// TwinCAT 3 PLC project SaftyPLC
// ProgramVersion: 3.1.4026.13
// libraries:
//   Tc2_Standard, * (Beckhoff Automation GmbH)
//   Tc2_System, * (Beckhoff Automation GmbH)
//   Tc2_Utilities, * (Beckhoff Automation GmbH)
//   Tc3_Module, * (Beckhoff Automation GmbH)
// project tree:
//   DUTs/GVLs/ GVL_IO.TcGVL, GVL_Safety.TcGVL (not stored)
//   / PlcTask.TcTTO (not stored)
//   POUs/ MAIN.TcPOU
// real-time tasks:
//   TASK XTS Task: cycle T#500us, priority 1, ADS port 350
//   TASK Job Task: cycle default, priority 32
//   TASK MC-Task (MET): cycle T#2ms, priority 3, ADS port 521
//   TASK MC-Task (MPT): cycle T#10ms, priority 8, ADS port 531
//   TASK PlcTask: cycle T#500us, priority 20, ADS port 351
// I/O:
//   DEVICE Device 8 (EtherCAT), AmsNetId 0.0.0.0.9.1
//     Box 23 (AT5100-0100) [AT5100-0100 XTS XL, TwinSAFE]
//       modules: Module 1 (SAFETY)
//     Box 24 (AT5100-0100) [AT5100-0100 XTS XL, TwinSAFE]
//       modules: Module 1 (SAFETY)
//     Box 25 (AT5100-0100) [AT5100-0100 XTS XL, TwinSAFE]
//       modules: Module 1 (SAFETY)
//     Box 26 (AT5100-0100) [AT5100-0100 XTS XL, TwinSAFE]
//       modules: Module 1 (SAFETY)
//     Box 27 (AT5100-0100) [AT5100-0100 XTS XL, TwinSAFE]
//       modules: Module 1 (SAFETY)
//     Box 28 (AT5100-0100) [AT5100-0100 XTS XL, TwinSAFE]
//       modules: Module 1 (SAFETY)
//     Box 29 (AT5100-0100) [AT5100-0100 XTS XL, TwinSAFE]
//       modules: Module 1 (SAFETY)
//     Box 30 (AT5100-0100) [AT5100-0100 XTS XL, TwinSAFE]
//       modules: Module 1 (SAFETY)
//     Box 31 (AT5100-0100) [AT5100-0100 XTS XL, TwinSAFE]
//       modules: Module 1 (SAFETY)
//     Box 32 (AT5100-0100) [AT5100-0100 XTS XL, TwinSAFE]
//       modules: Module 1 (SAFETY)
//     Box 33 (AT5100-0100) [AT5100-0100 XTS XL, TwinSAFE]
//       modules: Module 1 (SAFETY)
//     Box 34 (AT5100-0100) [AT5100-0100 XTS XL, TwinSAFE]
//       modules: Module 1 (SAFETY)
//     Box 35 (AT5100-0100) [AT5100-0100 XTS XL, TwinSAFE]
//       modules: Module 1 (SAFETY)
//     Box 36 (AT5100-0100) [AT5100-0100 XTS XL, TwinSAFE]
//       modules: Module 1 (SAFETY)
//     Box 37 (AT5100-0100) [AT5100-0100 XTS XL, TwinSAFE]
//       modules: Module 1 (SAFETY)
//     Box 38 (AT5100-0100) [AT5100-0100 XTS XL, TwinSAFE]
//       modules: Module 1 (SAFETY)
//     Box 39 (AT5100-0100) [AT5100-0100 XTS XL, TwinSAFE]
//       modules: Module 1 (SAFETY)
//     Box 40 (AT5100-0100) [AT5100-0100 XTS XL, TwinSAFE]
//       modules: Module 1 (SAFETY)
//     Box 41 (AT5100-0100) [AT5100-0100 XTS XL, TwinSAFE]
//       modules: Module 1 (SAFETY)
//     Box 42 (AT5100-0100) [AT5100-0100 XTS XL, TwinSAFE]
//       modules: Module 1 (SAFETY)
//     Box 43 (AT5100-0100) [AT5100-0100 XTS XL, TwinSAFE]
//       modules: Module 1 (SAFETY)
//     Box 44 (AT5100-0100) [AT5100-0100 XTS XL, TwinSAFE]
//       modules: Module 1 (SAFETY)
//     Box 45 (AT5100-0100) [AT5100-0100 XTS XL, TwinSAFE]
//       modules: Module 1 (SAFETY)
//     Box 46 (AT5100-0100) [AT5100-0100 XTS XL, TwinSAFE]
//       modules: Module 1 (SAFETY)
//     Box 47 (AT5100-0100) [AT5100-0100 XTS XL, TwinSAFE]
//       modules: Module 1 (SAFETY)
//     Box 48 (AT5100-0100) [AT5100-0100 XTS XL, TwinSAFE]
//       modules: Module 1 (SAFETY)
//     Box 49 (AT5100-0100) [AT5100-0100 XTS XL, TwinSAFE]
//       modules: Module 1 (SAFETY)
//   DEVICE Device 4 (EtherCAT), AmsNetId 0.0.0.0.5.1
//     Box 50 (AT5100-0100) [AT5100-0100 XTS XL, TwinSAFE]
//       modules: Module 1 (SAFETY)
//     Box 51 (AT5100-0100) [AT5100-0100 XTS XL, TwinSAFE]
//       modules: Module 1 (SAFETY)
//     Box 52 (AT5100-0100) [AT5100-0100 XTS XL, TwinSAFE]
//       modules: Module 1 (SAFETY)
//     Box 53 (AT5100-0100) [AT5100-0100 XTS XL, TwinSAFE]
//       modules: Module 1 (SAFETY)
//     Box 54 (AT5100-0100) [AT5100-0100 XTS XL, TwinSAFE]
//       modules: Module 1 (SAFETY)
//     Box 55 (AT5100-0100) [AT5100-0100 XTS XL, TwinSAFE]
//       modules: Module 1 (SAFETY)
//     Box 56 (AT5100-0100) [AT5100-0100 XTS XL, TwinSAFE]
//       modules: Module 1 (SAFETY)
//     Box 57 (AT5100-0100) [AT5100-0100 XTS XL, TwinSAFE]
//       modules: Module 1 (SAFETY)
//     Box 58 (AT5100-0100) [AT5100-0100 XTS XL, TwinSAFE]
//       modules: Module 1 (SAFETY)
//     Box 59 (AT5100-0100) [AT5100-0100 XTS XL, TwinSAFE]
//       modules: Module 1 (SAFETY)
//     Box 60 (AT5100-0100) [AT5100-0100 XTS XL, TwinSAFE]
//       modules: Module 1 (SAFETY)
//     Box 61 (AT5100-0100) [AT5100-0100 XTS XL, TwinSAFE]
//       modules: Module 1 (SAFETY)
//     Box 62 (AT5100-0100) [AT5100-0100 XTS XL, TwinSAFE]
//       modules: Module 1 (SAFETY)
//     Box 63 (AT5100-0100) [AT5100-0100 XTS XL, TwinSAFE]
//       modules: Module 1 (SAFETY)
//     Box 64 (AT5100-0100) [AT5100-0100 XTS XL, TwinSAFE]
//       modules: Module 1 (SAFETY)
//     Box 65 (AT5100-0100) [AT5100-0100 XTS XL, TwinSAFE]
//       modules: Module 1 (SAFETY)
//     Box 66 (AT5100-0100) [AT5100-0100 XTS XL, TwinSAFE]
//       modules: Module 1 (SAFETY)
//     Box 67 (AT5100-0100) [AT5100-0100 XTS XL, TwinSAFE]
//       modules: Module 1 (SAFETY)
//     Box 68 (AT5100-0100) [AT5100-0100 XTS XL, TwinSAFE]
//       modules: Module 1 (SAFETY)
//     Box 69 (AT5100-0100) [AT5100-0100 XTS XL, TwinSAFE]
//       modules: Module 1 (SAFETY)
//     Box 70 (AT5100-0100) [AT5100-0100 XTS XL, TwinSAFE]
//       modules: Module 1 (SAFETY)
//     Box 71 (AT5100-0100) [AT5100-0100 XTS XL, TwinSAFE]
//       modules: Module 1 (SAFETY)
//     Box 72 (AT5100-0100) [AT5100-0100 XTS XL, TwinSAFE]
//       modules: Module 1 (SAFETY)
//     Box 73 (AT5100-0100) [AT5100-0100 XTS XL, TwinSAFE]
//       modules: Module 1 (SAFETY)
//     Box 74 (AT5100-0100) [AT5100-0100 XTS XL, TwinSAFE]
//       modules: Module 1 (SAFETY)
//     Box 75 (AT5100-0100) [AT5100-0100 XTS XL, TwinSAFE]
//       modules: Module 1 (SAFETY)
//     Box 76 (AT5100-0100) [AT5100-0100 XTS XL, TwinSAFE]
//       modules: Module 1 (SAFETY)
//     Box 100 (AT5100-0100) [AT5100-0100 XTS XL, TwinSAFE]
//       modules: Module 1 (SAFETY)
//   DEVICE Device 1, AmsNetId 0.0.0.0.2.1
//     Term 1 (EK1200) [EK1200-5000 EtherCAT Power supply (2A E-Bus)]
//       Term 4 (EL1809) [EL1809 16Ch. Dig. Input 24V, 3ms]
//       Term 5 (EL1018) [EL1018 8Ch. Dig. Input 24V, 10µs]
//       Term 14 (EL2809) [EL2809 16Ch. Dig. Output 24V, 0.5A]
//       Term 17 (EL3004) [EL3004 4Ch. Ana. Input +/-10V]
//       Term 83 (EL3314) [EL3314 4Ch. Ana. Input Thermocouple (TC)]
//       Term 85 (EL4034) [EL4034 4Ch. Ana. Output +/-10V, 12bit]
//       Term 86 (EL7062) [EL7062-0000 Stepper Drive]
//       Term 87 (EL9576) [EL9576 Brake chopper terminal]
//       Term 88 (EL9410) [EL9410 E-Bus Power Supplier  (Diagnostics)]
//       Term 89 (EL1904) [EL1904, 4 Ch. Safety Input 24V, TwinSAFE]
//         modules: Module 1 (FSOES)
//       Term 90 (EL1904) [EL1904, 4 Ch. Safety Input 24V, TwinSAFE]
//         modules: Module 1 (FSOES)
//       Term 91 (EL2912) [EL2912, 2Ch. Safety Output 24V, 2A, TwinSAFE]
//         modules: Module 2 (FSOUT), Module 3 (DEVICEIO), Module 4 (FSLOGIC)
//       Term 92 (EK1110) [EK1110 EtherCAT extension]
//     Term 93 (AX8640-0000-0105) [AX8640-0000-0105] (disabled)
//       startup 32768:16 := 12 // PSM Parameters / Ext brake resistor overload factor at 1% duty cycle
//       startup 32768:18 := 21DCC63E // PSM Parameters / External brake resistor time constant 1
//       startup 32768:19 := C37C6442 // PSM Parameters / External brake resistor time constant 2
//       startup 32768:20 := 8CA3E13F // PSM Parameters / External brake resistor partial fraction factor
//   DEVICE Device 3 (EtherCAT Automation Protocol), AmsNetId 0.0.0.0.4.1
//     Box 28 (Publisher)
//     Box 29 (Subscriber)
//   DEVICE Device 5 (EtherCAT), AmsNetId 0.0.0.0.6.1
//     Box 1 (AT5840-0000) [AT5840-0000 Stromversorgung (300 V, 16 A, 3-phasig)]
// variable links:
//   Device 1 <-> Device 1/Term 1 (EK1200)/Term 90 (EL1904)
//     Term 1 (EK1200)/Term 91 (EL2912)/ConnectionInputs/Message_142 TxPDO <-> Module 1 (FSOES)/RxPDO/FSOE
//   Device 1 <-> Device 1/Term 1 (EK1200)/Term 91 (EL2912)
//     Term 1 (EK1200)/Term 89 (EL1904)/Module 1 (FSOES)/RxPDO/FSOE <-> ConnectionInputs/Message_141 TxPDO
//     Term 1 (EK1200)/Term 89 (EL1904)/Module 1 (FSOES)/TxPDO/FSOE <-> ConnectionOutputs/Message_141 RxPDO
//     Term 1 (EK1200)/Term 90 (EL1904)/Module 1 (FSOES)/TxPDO/FSOE <-> ConnectionOutputs/Message_142 RxPDO
//   Device 1 <-> Device 3 (EtherCAT Automation Protocol)/Box 28 (Publisher)
//     Term 1 (EK1200)/Term 91 (EL2912)/ConnectionInputs/Message_143 TxPDO <-> Safety/Outputs/VarData
//   Device 1 <-> Device 3 (EtherCAT Automation Protocol)/Box 29 (Subscriber)
//     Term 1 (EK1200)/Term 91 (EL2912)/ConnectionOutputs/Message_143 RxPDO <-> Safety/Inputs/VarData
//   Device 1 <-> Device 4 (EtherCAT)/Box 63 (AT5100-0100)
//     Term 1 (EK1200)/Term 91 (EL2912)/ConnectionInputs/Message_120 TxPDO <-> Module 1 (SAFETY)/SAFETY FSoE Connection 1 Receive Message/Message_4
//   Device 1 <-> Device 8 (EtherCAT)/Box 30 (AT5100-0100)
//     Term 1 (EK1200)/Term 91 (EL2912)/ConnectionOutputs/Message_87 RxPDO <-> Module 1 (SAFETY)/SAFETY FSoE Connection 1 Send Message/Message_4
//   Device 4 (EtherCAT) <-> Device 1/Term 1 (EK1200)/Term 91 (EL2912)
//     Box 50 (AT5100-0100)/Module 1 (SAFETY)/SAFETY FSoE Connection 1 Receive Message/Message_4 <-> ConnectionInputs/Message_107 TxPDO
//     Box 51 (AT5100-0100)/Module 1 (SAFETY)/SAFETY FSoE Connection 1 Receive Message/Message_4 <-> ConnectionInputs/Message_108 TxPDO
//     Box 52 (AT5100-0100)/Module 1 (SAFETY)/SAFETY FSoE Connection 1 Receive Message/Message_4 <-> ConnectionInputs/Message_109 TxPDO
//     Box 53 (AT5100-0100)/Module 1 (SAFETY)/SAFETY FSoE Connection 1 Receive Message/Message_4 <-> ConnectionInputs/Message_110 TxPDO
//     Box 54 (AT5100-0100)/Module 1 (SAFETY)/SAFETY FSoE Connection 1 Receive Message/Message_4 <-> ConnectionInputs/Message_111 TxPDO
//     Box 55 (AT5100-0100)/Module 1 (SAFETY)/SAFETY FSoE Connection 1 Receive Message/Message_4 <-> ConnectionInputs/Message_112 TxPDO
//     Box 56 (AT5100-0100)/Module 1 (SAFETY)/SAFETY FSoE Connection 1 Receive Message/Message_4 <-> ConnectionInputs/Message_113 TxPDO
//     Box 57 (AT5100-0100)/Module 1 (SAFETY)/SAFETY FSoE Connection 1 Receive Message/Message_4 <-> ConnectionInputs/Message_114 TxPDO
//     Box 58 (AT5100-0100)/Module 1 (SAFETY)/SAFETY FSoE Connection 1 Receive Message/Message_4 <-> ConnectionInputs/Message_115 TxPDO
//     Box 59 (AT5100-0100)/Module 1 (SAFETY)/SAFETY FSoE Connection 1 Receive Message/Message_4 <-> ConnectionInputs/Message_116 TxPDO
//     Box 60 (AT5100-0100)/Module 1 (SAFETY)/SAFETY FSoE Connection 1 Receive Message/Message_4 <-> ConnectionInputs/Message_117 TxPDO
//     Box 61 (AT5100-0100)/Module 1 (SAFETY)/SAFETY FSoE Connection 1 Receive Message/Message_4 <-> ConnectionInputs/Message_118 TxPDO
//     Box 62 (AT5100-0100)/Module 1 (SAFETY)/SAFETY FSoE Connection 1 Receive Message/Message_4 <-> ConnectionInputs/Message_119 TxPDO
//     Box 64 (AT5100-0100)/Module 1 (SAFETY)/SAFETY FSoE Connection 1 Receive Message/Message_4 <-> ConnectionInputs/Message_121 TxPDO
//     Box 65 (AT5100-0100)/Module 1 (SAFETY)/SAFETY FSoE Connection 1 Receive Message/Message_4 <-> ConnectionInputs/Message_122 TxPDO
//     Box 66 (AT5100-0100)/Module 1 (SAFETY)/SAFETY FSoE Connection 1 Receive Message/Message_4 <-> ConnectionInputs/Message_123 TxPDO
//     Box 67 (AT5100-0100)/Module 1 (SAFETY)/SAFETY FSoE Connection 1 Receive Message/Message_4 <-> ConnectionInputs/Message_124 TxPDO
//     Box 68 (AT5100-0100)/Module 1 (SAFETY)/SAFETY FSoE Connection 1 Receive Message/Message_4 <-> ConnectionInputs/Message_125 TxPDO
//     Box 69 (AT5100-0100)/Module 1 (SAFETY)/SAFETY FSoE Connection 1 Receive Message/Message_4 <-> ConnectionInputs/Message_126 TxPDO
//     Box 70 (AT5100-0100)/Module 1 (SAFETY)/SAFETY FSoE Connection 1 Receive Message/Message_4 <-> ConnectionInputs/Message_127 TxPDO
//     Box 71 (AT5100-0100)/Module 1 (SAFETY)/SAFETY FSoE Connection 1 Receive Message/Message_4 <-> ConnectionInputs/Message_128 TxPDO
//     Box 72 (AT5100-0100)/Module 1 (SAFETY)/SAFETY FSoE Connection 1 Receive Message/Message_4 <-> ConnectionInputs/Message_129 TxPDO
//     Box 73 (AT5100-0100)/Module 1 (SAFETY)/SAFETY FSoE Connection 1 Receive Message/Message_4 <-> ConnectionInputs/Message_130 TxPDO
//     Box 74 (AT5100-0100)/Module 1 (SAFETY)/SAFETY FSoE Connection 1 Receive Message/Message_4 <-> ConnectionInputs/Message_131 TxPDO
//     Box 75 (AT5100-0100)/Module 1 (SAFETY)/SAFETY FSoE Connection 1 Receive Message/Message_4 <-> ConnectionInputs/Message_132 TxPDO
//     Box 76 (AT5100-0100)/Module 1 (SAFETY)/SAFETY FSoE Connection 1 Receive Message/Message_4 <-> ConnectionInputs/Message_133 TxPDO
//     Box 50 (AT5100-0100)/Module 1 (SAFETY)/SAFETY FSoE Connection 1 Send Message/Message_4 <-> ConnectionOutputs/Message_107 RxPDO
//     Box 51 (AT5100-0100)/Module 1 (SAFETY)/SAFETY FSoE Connection 1 Send Message/Message_4 <-> ConnectionOutputs/Message_108 RxPDO
//     Box 52 (AT5100-0100)/Module 1 (SAFETY)/SAFETY FSoE Connection 1 Send Message/Message_4 <-> ConnectionOutputs/Message_109 RxPDO
//     Box 53 (AT5100-0100)/Module 1 (SAFETY)/SAFETY FSoE Connection 1 Send Message/Message_4 <-> ConnectionOutputs/Message_110 RxPDO
//     Box 54 (AT5100-0100)/Module 1 (SAFETY)/SAFETY FSoE Connection 1 Send Message/Message_4 <-> ConnectionOutputs/Message_111 RxPDO
//     Box 55 (AT5100-0100)/Module 1 (SAFETY)/SAFETY FSoE Connection 1 Send Message/Message_4 <-> ConnectionOutputs/Message_112 RxPDO
//     Box 56 (AT5100-0100)/Module 1 (SAFETY)/SAFETY FSoE Connection 1 Send Message/Message_4 <-> ConnectionOutputs/Message_113 RxPDO
//     Box 57 (AT5100-0100)/Module 1 (SAFETY)/SAFETY FSoE Connection 1 Send Message/Message_4 <-> ConnectionOutputs/Message_114 RxPDO
//     Box 58 (AT5100-0100)/Module 1 (SAFETY)/SAFETY FSoE Connection 1 Send Message/Message_4 <-> ConnectionOutputs/Message_115 RxPDO
//     Box 59 (AT5100-0100)/Module 1 (SAFETY)/SAFETY FSoE Connection 1 Send Message/Message_4 <-> ConnectionOutputs/Message_116 RxPDO
//     Box 60 (AT5100-0100)/Module 1 (SAFETY)/SAFETY FSoE Connection 1 Send Message/Message_4 <-> ConnectionOutputs/Message_117 RxPDO
//     Box 61 (AT5100-0100)/Module 1 (SAFETY)/SAFETY FSoE Connection 1 Send Message/Message_4 <-> ConnectionOutputs/Message_118 RxPDO
//     Box 62 (AT5100-0100)/Module 1 (SAFETY)/SAFETY FSoE Connection 1 Send Message/Message_4 <-> ConnectionOutputs/Message_119 RxPDO
//     Box 63 (AT5100-0100)/Module 1 (SAFETY)/SAFETY FSoE Connection 1 Send Message/Message_4 <-> ConnectionOutputs/Message_120 RxPDO
//     Box 64 (AT5100-0100)/Module 1 (SAFETY)/SAFETY FSoE Connection 1 Send Message/Message_4 <-> ConnectionOutputs/Message_121 RxPDO
//     Box 65 (AT5100-0100)/Module 1 (SAFETY)/SAFETY FSoE Connection 1 Send Message/Message_4 <-> ConnectionOutputs/Message_122 RxPDO
//     Box 66 (AT5100-0100)/Module 1 (SAFETY)/SAFETY FSoE Connection 1 Send Message/Message_4 <-> ConnectionOutputs/Message_123 RxPDO
//     Box 67 (AT5100-0100)/Module 1 (SAFETY)/SAFETY FSoE Connection 1 Send Message/Message_4 <-> ConnectionOutputs/Message_124 RxPDO
//     Box 68 (AT5100-0100)/Module 1 (SAFETY)/SAFETY FSoE Connection 1 Send Message/Message_4 <-> ConnectionOutputs/Message_125 RxPDO
//     Box 69 (AT5100-0100)/Module 1 (SAFETY)/SAFETY FSoE Connection 1 Send Message/Message_4 <-> ConnectionOutputs/Message_126 RxPDO
//     Box 70 (AT5100-0100)/Module 1 (SAFETY)/SAFETY FSoE Connection 1 Send Message/Message_4 <-> ConnectionOutputs/Message_127 RxPDO
//     Box 71 (AT5100-0100)/Module 1 (SAFETY)/SAFETY FSoE Connection 1 Send Message/Message_4 <-> ConnectionOutputs/Message_128 RxPDO
//     Box 72 (AT5100-0100)/Module 1 (SAFETY)/SAFETY FSoE Connection 1 Send Message/Message_4 <-> ConnectionOutputs/Message_129 RxPDO
//     Box 73 (AT5100-0100)/Module 1 (SAFETY)/SAFETY FSoE Connection 1 Send Message/Message_4 <-> ConnectionOutputs/Message_130 RxPDO
//     Box 74 (AT5100-0100)/Module 1 (SAFETY)/SAFETY FSoE Connection 1 Send Message/Message_4 <-> ConnectionOutputs/Message_131 RxPDO
//     Box 75 (AT5100-0100)/Module 1 (SAFETY)/SAFETY FSoE Connection 1 Send Message/Message_4 <-> ConnectionOutputs/Message_132 RxPDO
//     Box 76 (AT5100-0100)/Module 1 (SAFETY)/SAFETY FSoE Connection 1 Send Message/Message_4 <-> ConnectionOutputs/Message_133 RxPDO
//   Device 8 (EtherCAT) <-> Device 1/Term 1 (EK1200)/Term 91 (EL2912)
//     Box 23 (AT5100-0100)/Module 1 (SAFETY)/SAFETY FSoE Connection 1 Receive Message/Message_4 <-> ConnectionInputs/Message_80 TxPDO
//     Box 24 (AT5100-0100)/Module 1 (SAFETY)/SAFETY FSoE Connection 1 Receive Message/Message_4 <-> ConnectionInputs/Message_81 TxPDO
//     Box 25 (AT5100-0100)/Module 1 (SAFETY)/SAFETY FSoE Connection 1 Receive Message/Message_4 <-> ConnectionInputs/Message_82 TxPDO
//     Box 26 (AT5100-0100)/Module 1 (SAFETY)/SAFETY FSoE Connection 1 Receive Message/Message_4 <-> ConnectionInputs/Message_83 TxPDO
//     Box 27 (AT5100-0100)/Module 1 (SAFETY)/SAFETY FSoE Connection 1 Receive Message/Message_4 <-> ConnectionInputs/Message_84 TxPDO
//     Box 28 (AT5100-0100)/Module 1 (SAFETY)/SAFETY FSoE Connection 1 Receive Message/Message_4 <-> ConnectionInputs/Message_85 TxPDO
//     Box 29 (AT5100-0100)/Module 1 (SAFETY)/SAFETY FSoE Connection 1 Receive Message/Message_4 <-> ConnectionInputs/Message_86 TxPDO
//     Box 30 (AT5100-0100)/Module 1 (SAFETY)/SAFETY FSoE Connection 1 Receive Message/Message_4 <-> ConnectionInputs/Message_87 TxPDO
//     Box 31 (AT5100-0100)/Module 1 (SAFETY)/SAFETY FSoE Connection 1 Receive Message/Message_4 <-> ConnectionInputs/Message_88 TxPDO
//     Box 32 (AT5100-0100)/Module 1 (SAFETY)/SAFETY FSoE Connection 1 Receive Message/Message_4 <-> ConnectionInputs/Message_89 TxPDO
//     Box 33 (AT5100-0100)/Module 1 (SAFETY)/SAFETY FSoE Connection 1 Receive Message/Message_4 <-> ConnectionInputs/Message_90 TxPDO
//     Box 34 (AT5100-0100)/Module 1 (SAFETY)/SAFETY FSoE Connection 1 Receive Message/Message_4 <-> ConnectionInputs/Message_91 TxPDO
//     Box 35 (AT5100-0100)/Module 1 (SAFETY)/SAFETY FSoE Connection 1 Receive Message/Message_4 <-> ConnectionInputs/Message_92 TxPDO
//     Box 36 (AT5100-0100)/Module 1 (SAFETY)/SAFETY FSoE Connection 1 Receive Message/Message_4 <-> ConnectionInputs/Message_93 TxPDO
//     Box 37 (AT5100-0100)/Module 1 (SAFETY)/SAFETY FSoE Connection 1 Receive Message/Message_4 <-> ConnectionInputs/Message_94 TxPDO
//     Box 38 (AT5100-0100)/Module 1 (SAFETY)/SAFETY FSoE Connection 1 Receive Message/Message_4 <-> ConnectionInputs/Message_95 TxPDO
//     Box 39 (AT5100-0100)/Module 1 (SAFETY)/SAFETY FSoE Connection 1 Receive Message/Message_4 <-> ConnectionInputs/Message_96 TxPDO
//     Box 40 (AT5100-0100)/Module 1 (SAFETY)/SAFETY FSoE Connection 1 Receive Message/Message_4 <-> ConnectionInputs/Message_97 TxPDO
//     Box 41 (AT5100-0100)/Module 1 (SAFETY)/SAFETY FSoE Connection 1 Receive Message/Message_4 <-> ConnectionInputs/Message_98 TxPDO
//     Box 42 (AT5100-0100)/Module 1 (SAFETY)/SAFETY FSoE Connection 1 Receive Message/Message_4 <-> ConnectionInputs/Message_99 TxPDO
//     Box 43 (AT5100-0100)/Module 1 (SAFETY)/SAFETY FSoE Connection 1 Receive Message/Message_4 <-> ConnectionInputs/Message_100 TxPDO
//     Box 44 (AT5100-0100)/Module 1 (SAFETY)/SAFETY FSoE Connection 1 Receive Message/Message_4 <-> ConnectionInputs/Message_101 TxPDO
//     Box 45 (AT5100-0100)/Module 1 (SAFETY)/SAFETY FSoE Connection 1 Receive Message/Message_4 <-> ConnectionInputs/Message_102 TxPDO
//     Box 46 (AT5100-0100)/Module 1 (SAFETY)/SAFETY FSoE Connection 1 Receive Message/Message_4 <-> ConnectionInputs/Message_103 TxPDO
//     Box 47 (AT5100-0100)/Module 1 (SAFETY)/SAFETY FSoE Connection 1 Receive Message/Message_4 <-> ConnectionInputs/Message_104 TxPDO
//     Box 48 (AT5100-0100)/Module 1 (SAFETY)/SAFETY FSoE Connection 1 Receive Message/Message_4 <-> ConnectionInputs/Message_105 TxPDO
//     Box 49 (AT5100-0100)/Module 1 (SAFETY)/SAFETY FSoE Connection 1 Receive Message/Message_4 <-> ConnectionInputs/Message_106 TxPDO
//     Box 23 (AT5100-0100)/Module 1 (SAFETY)/SAFETY FSoE Connection 1 Send Message/Message_4 <-> ConnectionOutputs/Message_80 RxPDO
//     Box 24 (AT5100-0100)/Module 1 (SAFETY)/SAFETY FSoE Connection 1 Send Message/Message_4 <-> ConnectionOutputs/Message_81 RxPDO
//     Box 25 (AT5100-0100)/Module 1 (SAFETY)/SAFETY FSoE Connection 1 Send Message/Message_4 <-> ConnectionOutputs/Message_82 RxPDO
//     Box 26 (AT5100-0100)/Module 1 (SAFETY)/SAFETY FSoE Connection 1 Send Message/Message_4 <-> ConnectionOutputs/Message_83 RxPDO
//     Box 27 (AT5100-0100)/Module 1 (SAFETY)/SAFETY FSoE Connection 1 Send Message/Message_4 <-> ConnectionOutputs/Message_84 RxPDO
//     Box 28 (AT5100-0100)/Module 1 (SAFETY)/SAFETY FSoE Connection 1 Send Message/Message_4 <-> ConnectionOutputs/Message_85 RxPDO
//     Box 29 (AT5100-0100)/Module 1 (SAFETY)/SAFETY FSoE Connection 1 Send Message/Message_4 <-> ConnectionOutputs/Message_86 RxPDO
//     Box 31 (AT5100-0100)/Module 1 (SAFETY)/SAFETY FSoE Connection 1 Send Message/Message_4 <-> ConnectionOutputs/Message_88 RxPDO
//     Box 32 (AT5100-0100)/Module 1 (SAFETY)/SAFETY FSoE Connection 1 Send Message/Message_4 <-> ConnectionOutputs/Message_89 RxPDO
//     Box 33 (AT5100-0100)/Module 1 (SAFETY)/SAFETY FSoE Connection 1 Send Message/Message_4 <-> ConnectionOutputs/Message_90 RxPDO
//     Box 34 (AT5100-0100)/Module 1 (SAFETY)/SAFETY FSoE Connection 1 Send Message/Message_4 <-> ConnectionOutputs/Message_91 RxPDO
//     Box 35 (AT5100-0100)/Module 1 (SAFETY)/SAFETY FSoE Connection 1 Send Message/Message_4 <-> ConnectionOutputs/Message_92 RxPDO
//     Box 36 (AT5100-0100)/Module 1 (SAFETY)/SAFETY FSoE Connection 1 Send Message/Message_4 <-> ConnectionOutputs/Message_93 RxPDO
//     Box 37 (AT5100-0100)/Module 1 (SAFETY)/SAFETY FSoE Connection 1 Send Message/Message_4 <-> ConnectionOutputs/Message_94 RxPDO
//     Box 38 (AT5100-0100)/Module 1 (SAFETY)/SAFETY FSoE Connection 1 Send Message/Message_4 <-> ConnectionOutputs/Message_95 RxPDO
//     Box 39 (AT5100-0100)/Module 1 (SAFETY)/SAFETY FSoE Connection 1 Send Message/Message_4 <-> ConnectionOutputs/Message_96 RxPDO
//     Box 40 (AT5100-0100)/Module 1 (SAFETY)/SAFETY FSoE Connection 1 Send Message/Message_4 <-> ConnectionOutputs/Message_97 RxPDO
//     Box 41 (AT5100-0100)/Module 1 (SAFETY)/SAFETY FSoE Connection 1 Send Message/Message_4 <-> ConnectionOutputs/Message_98 RxPDO
//     Box 42 (AT5100-0100)/Module 1 (SAFETY)/SAFETY FSoE Connection 1 Send Message/Message_4 <-> ConnectionOutputs/Message_99 RxPDO
//     Box 43 (AT5100-0100)/Module 1 (SAFETY)/SAFETY FSoE Connection 1 Send Message/Message_4 <-> ConnectionOutputs/Message_100 RxPDO
//     Box 44 (AT5100-0100)/Module 1 (SAFETY)/SAFETY FSoE Connection 1 Send Message/Message_4 <-> ConnectionOutputs/Message_101 RxPDO
//     Box 45 (AT5100-0100)/Module 1 (SAFETY)/SAFETY FSoE Connection 1 Send Message/Message_4 <-> ConnectionOutputs/Message_102 RxPDO
//     Box 46 (AT5100-0100)/Module 1 (SAFETY)/SAFETY FSoE Connection 1 Send Message/Message_4 <-> ConnectionOutputs/Message_103 RxPDO
//     Box 47 (AT5100-0100)/Module 1 (SAFETY)/SAFETY FSoE Connection 1 Send Message/Message_4 <-> ConnectionOutputs/Message_104 RxPDO
//     Box 48 (AT5100-0100)/Module 1 (SAFETY)/SAFETY FSoE Connection 1 Send Message/Message_4 <-> ConnectionOutputs/Message_105 RxPDO
//     Box 49 (AT5100-0100)/Module 1 (SAFETY)/SAFETY FSoE Connection 1 Send Message/Message_4 <-> ConnectionOutputs/Message_106 RxPDO
//   MC3_Multi_IPC1/MC3_Multi_IPC1 Instance <-> Device 1/Term 1 (EK1200)/Term 85 (EL4034)
//     PlcTask Outputs/MAIN_S1.MagnetValue <-> AO Outputs Channel 1/Analog output
//   MC3_Multi_IPC1/MC3_Multi_IPC1 Instance <-> Device 3 (EtherCAT Automation Protocol)/Box 28 (Publisher)
//     PlcTask Outputs/GVL_DataExchange.Dynamics <-> Command/Outputs/VarData/Dynamics
//   MC3_Multi_IPC1/MC3_Multi_IPC1 Instance <-> MC Project IPC1/Axes/MC_Mover 1
//     PlcTask Inputs/GVL_MC.fbMover[1].fbPlanarMover.MCTOPLC/ACT <-> McToPlc/ACT
//     PlcTask Inputs/GVL_MC.fbMover[1].fbPlanarMover.MCTOPLC/COORDMODE <-> McToPlc/COORDMODE
//     PlcTask Inputs/GVL_MC.fbMover[1].fbPlanarMover.MCTOPLC/SET <-> McToPlc/SET
//     PlcTask Inputs/GVL_MC.fbMover[1].fbPlanarMover.MCTOPLC/SETONTRACK <-> McToPlc/SETONTRACK
//     PlcTask Inputs/GVL_MC.fbMover[1].fbPlanarMover.MCTOPLC/STD <-> McToPlc/STD
//     PlcTask Outputs/GVL_MC.fbMover[1].fbPlanarMover.PLCTOMC/STD <-> PlcToMc/STD
//   MC3_Multi_IPC1/MC3_Multi_IPC1 Instance <-> MC Project IPC1/Axes/MC_Mover 10
//     PlcTask Inputs/GVL_MC.fbMover[10].fbPlanarMover.MCTOPLC/ACT <-> McToPlc/ACT
//     PlcTask Inputs/GVL_MC.fbMover[10].fbPlanarMover.MCTOPLC/COORDMODE <-> McToPlc/COORDMODE
//     PlcTask Inputs/GVL_MC.fbMover[10].fbPlanarMover.MCTOPLC/SET <-> McToPlc/SET
//     PlcTask Inputs/GVL_MC.fbMover[10].fbPlanarMover.MCTOPLC/SETONTRACK <-> McToPlc/SETONTRACK
//     PlcTask Inputs/GVL_MC.fbMover[10].fbPlanarMover.MCTOPLC/STD <-> McToPlc/STD
//     PlcTask Outputs/GVL_MC.fbMover[10].fbPlanarMover.PLCTOMC/STD <-> PlcToMc/STD
//   MC3_Multi_IPC1/MC3_Multi_IPC1 Instance <-> MC Project IPC1/Axes/MC_Mover 11
//     PlcTask Inputs/GVL_MC.fbMover[11].fbPlanarMover.MCTOPLC/ACT <-> McToPlc/ACT
//     PlcTask Inputs/GVL_MC.fbMover[11].fbPlanarMover.MCTOPLC/COORDMODE <-> McToPlc/COORDMODE
//     PlcTask Inputs/GVL_MC.fbMover[11].fbPlanarMover.MCTOPLC/SET <-> McToPlc/SET
//     PlcTask Inputs/GVL_MC.fbMover[11].fbPlanarMover.MCTOPLC/SETONTRACK <-> McToPlc/SETONTRACK
//     PlcTask Inputs/GVL_MC.fbMover[11].fbPlanarMover.MCTOPLC/STD <-> McToPlc/STD
//     PlcTask Outputs/GVL_MC.fbMover[11].fbPlanarMover.PLCTOMC/STD <-> PlcToMc/STD
//   MC3_Multi_IPC1/MC3_Multi_IPC1 Instance <-> MC Project IPC1/Axes/MC_Mover 12
//     PlcTask Inputs/GVL_MC.fbMover[12].fbPlanarMover.MCTOPLC/ACT <-> McToPlc/ACT
//     PlcTask Inputs/GVL_MC.fbMover[12].fbPlanarMover.MCTOPLC/COORDMODE <-> McToPlc/COORDMODE
//     PlcTask Inputs/GVL_MC.fbMover[12].fbPlanarMover.MCTOPLC/SET <-> McToPlc/SET
//     PlcTask Inputs/GVL_MC.fbMover[12].fbPlanarMover.MCTOPLC/SETONTRACK <-> McToPlc/SETONTRACK
//     PlcTask Inputs/GVL_MC.fbMover[12].fbPlanarMover.MCTOPLC/STD <-> McToPlc/STD
//     PlcTask Outputs/GVL_MC.fbMover[12].fbPlanarMover.PLCTOMC/STD <-> PlcToMc/STD
//   MC3_Multi_IPC1/MC3_Multi_IPC1 Instance <-> MC Project IPC1/Axes/MC_Mover 2
//     PlcTask Inputs/GVL_MC.fbMover[2].fbPlanarMover.MCTOPLC/ACT <-> McToPlc/ACT
//     PlcTask Inputs/GVL_MC.fbMover[2].fbPlanarMover.MCTOPLC/COORDMODE <-> McToPlc/COORDMODE
//     PlcTask Inputs/GVL_MC.fbMover[2].fbPlanarMover.MCTOPLC/SET <-> McToPlc/SET
//     PlcTask Inputs/GVL_MC.fbMover[2].fbPlanarMover.MCTOPLC/SETONTRACK <-> McToPlc/SETONTRACK
//     PlcTask Inputs/GVL_MC.fbMover[2].fbPlanarMover.MCTOPLC/STD <-> McToPlc/STD
//     PlcTask Outputs/GVL_MC.fbMover[2].fbPlanarMover.PLCTOMC/STD <-> PlcToMc/STD
//   MC3_Multi_IPC1/MC3_Multi_IPC1 Instance <-> MC Project IPC1/Axes/MC_Mover 3
//     PlcTask Inputs/GVL_MC.fbMover[3].fbPlanarMover.MCTOPLC/ACT <-> McToPlc/ACT
//     PlcTask Inputs/GVL_MC.fbMover[3].fbPlanarMover.MCTOPLC/COORDMODE <-> McToPlc/COORDMODE
//     PlcTask Inputs/GVL_MC.fbMover[3].fbPlanarMover.MCTOPLC/SET <-> McToPlc/SET
//     PlcTask Inputs/GVL_MC.fbMover[3].fbPlanarMover.MCTOPLC/SETONTRACK <-> McToPlc/SETONTRACK
//     PlcTask Inputs/GVL_MC.fbMover[3].fbPlanarMover.MCTOPLC/STD <-> McToPlc/STD
//     PlcTask Outputs/GVL_MC.fbMover[3].fbPlanarMover.PLCTOMC/STD <-> PlcToMc/STD
//   MC3_Multi_IPC1/MC3_Multi_IPC1 Instance <-> MC Project IPC1/Axes/MC_Mover 4
//     PlcTask Inputs/GVL_MC.fbMover[4].fbPlanarMover.MCTOPLC/ACT <-> McToPlc/ACT
//     PlcTask Inputs/GVL_MC.fbMover[4].fbPlanarMover.MCTOPLC/COORDMODE <-> McToPlc/COORDMODE
//     PlcTask Inputs/GVL_MC.fbMover[4].fbPlanarMover.MCTOPLC/SET <-> McToPlc/SET
//     PlcTask Inputs/GVL_MC.fbMover[4].fbPlanarMover.MCTOPLC/SETONTRACK <-> McToPlc/SETONTRACK
//     PlcTask Inputs/GVL_MC.fbMover[4].fbPlanarMover.MCTOPLC/STD <-> McToPlc/STD
//     PlcTask Outputs/GVL_MC.fbMover[4].fbPlanarMover.PLCTOMC/STD <-> PlcToMc/STD
//   MC3_Multi_IPC1/MC3_Multi_IPC1 Instance <-> MC Project IPC1/Axes/MC_Mover 5
//     PlcTask Inputs/GVL_MC.fbMover[5].fbPlanarMover.MCTOPLC/ACT <-> McToPlc/ACT
//     PlcTask Inputs/GVL_MC.fbMover[5].fbPlanarMover.MCTOPLC/COORDMODE <-> McToPlc/COORDMODE
//     PlcTask Inputs/GVL_MC.fbMover[5].fbPlanarMover.MCTOPLC/SET <-> McToPlc/SET
//     PlcTask Inputs/GVL_MC.fbMover[5].fbPlanarMover.MCTOPLC/SETONTRACK <-> McToPlc/SETONTRACK
//     PlcTask Inputs/GVL_MC.fbMover[5].fbPlanarMover.MCTOPLC/STD <-> McToPlc/STD
//     PlcTask Outputs/GVL_MC.fbMover[5].fbPlanarMover.PLCTOMC/STD <-> PlcToMc/STD
//   MC3_Multi_IPC1/MC3_Multi_IPC1 Instance <-> MC Project IPC1/Axes/MC_Mover 6
//     PlcTask Inputs/GVL_MC.fbMover[6].fbPlanarMover.MCTOPLC/ACT <-> McToPlc/ACT
//     PlcTask Inputs/GVL_MC.fbMover[6].fbPlanarMover.MCTOPLC/COORDMODE <-> McToPlc/COORDMODE
//     PlcTask Inputs/GVL_MC.fbMover[6].fbPlanarMover.MCTOPLC/SET <-> McToPlc/SET
//     PlcTask Inputs/GVL_MC.fbMover[6].fbPlanarMover.MCTOPLC/SETONTRACK <-> McToPlc/SETONTRACK
//     PlcTask Inputs/GVL_MC.fbMover[6].fbPlanarMover.MCTOPLC/STD <-> McToPlc/STD
//     PlcTask Outputs/GVL_MC.fbMover[6].fbPlanarMover.PLCTOMC/STD <-> PlcToMc/STD
//   MC3_Multi_IPC1/MC3_Multi_IPC1 Instance <-> MC Project IPC1/Axes/MC_Mover 7
//     PlcTask Inputs/GVL_MC.fbMover[7].fbPlanarMover.MCTOPLC/ACT <-> McToPlc/ACT
//     PlcTask Inputs/GVL_MC.fbMover[7].fbPlanarMover.MCTOPLC/COORDMODE <-> McToPlc/COORDMODE
//     PlcTask Inputs/GVL_MC.fbMover[7].fbPlanarMover.MCTOPLC/SET <-> McToPlc/SET
//     PlcTask Inputs/GVL_MC.fbMover[7].fbPlanarMover.MCTOPLC/SETONTRACK <-> McToPlc/SETONTRACK
//     PlcTask Inputs/GVL_MC.fbMover[7].fbPlanarMover.MCTOPLC/STD <-> McToPlc/STD
//     PlcTask Outputs/GVL_MC.fbMover[7].fbPlanarMover.PLCTOMC/STD <-> PlcToMc/STD
//   MC3_Multi_IPC1/MC3_Multi_IPC1 Instance <-> MC Project IPC1/Axes/MC_Mover 8
//     PlcTask Inputs/GVL_MC.fbMover[8].fbPlanarMover.MCTOPLC/ACT <-> McToPlc/ACT
//     PlcTask Inputs/GVL_MC.fbMover[8].fbPlanarMover.MCTOPLC/COORDMODE <-> McToPlc/COORDMODE
//     PlcTask Inputs/GVL_MC.fbMover[8].fbPlanarMover.MCTOPLC/SET <-> McToPlc/SET
//     PlcTask Inputs/GVL_MC.fbMover[8].fbPlanarMover.MCTOPLC/SETONTRACK <-> McToPlc/SETONTRACK
//     PlcTask Inputs/GVL_MC.fbMover[8].fbPlanarMover.MCTOPLC/STD <-> McToPlc/STD
//     PlcTask Outputs/GVL_MC.fbMover[8].fbPlanarMover.PLCTOMC/STD <-> PlcToMc/STD
//   MC3_Multi_IPC1/MC3_Multi_IPC1 Instance <-> MC Project IPC1/Axes/MC_Mover 9
//     PlcTask Inputs/GVL_MC.fbMover[9].fbPlanarMover.MCTOPLC/ACT <-> McToPlc/ACT
//     PlcTask Inputs/GVL_MC.fbMover[9].fbPlanarMover.MCTOPLC/COORDMODE <-> McToPlc/COORDMODE
//     PlcTask Inputs/GVL_MC.fbMover[9].fbPlanarMover.MCTOPLC/SET <-> McToPlc/SET
//     PlcTask Inputs/GVL_MC.fbMover[9].fbPlanarMover.MCTOPLC/SETONTRACK <-> McToPlc/SETONTRACK
//     PlcTask Inputs/GVL_MC.fbMover[9].fbPlanarMover.MCTOPLC/STD <-> McToPlc/STD
//     PlcTask Outputs/GVL_MC.fbMover[9].fbPlanarMover.PLCTOMC/STD <-> PlcToMc/STD
//   MC3_Multi_IPC1/MC3_Multi_IPC1 Instance <-> MC Project IPC1/Groups/IPC 1 In Connection
//     PlcTask Inputs/GVL_MC.EnterSystem.MCTOPLC_STD <-> McToPlc/STD
//   MC3_Multi_IPC1/MC3_Multi_IPC1 Instance <-> MC Project IPC1/Groups/IPC 1 Out Connection
//     PlcTask Inputs/GVL_MC.ExitSystem.MCTOPLC_STD <-> McToPlc/STD
//   MC3_Multi_IPC1/MC3_Multi_IPC1 Instance <-> MC Project IPC1/Groups/McTrack1
//     PlcTask Inputs/GVL_MC.aMcTracks[2].MCTOPLC_STD <-> McToPlc/STD
//   MC3_Multi_IPC1/MC3_Multi_IPC1 Instance <-> MC Project IPC1/Groups/McTrack2
//     PlcTask Inputs/GVL_MC.aMcTracks[4].MCTOPLC_STD <-> McToPlc/STD
//   MC3_Multi_IPC1/MC3_Multi_IPC1 Instance <-> MC Project IPC1/Groups/McTrack3.1 Start
//     PlcTask Inputs/GVL_MC.aMcTracks[1].MCTOPLC_STD <-> McToPlc/STD
//   MC3_Multi_IPC1/MC3_Multi_IPC1 Instance <-> MC Project IPC1/Groups/McTrack3.2 End
//     PlcTask Inputs/GVL_MC.aMcTracks[3].MCTOPLC_STD <-> McToPlc/STD
//   SaftyPLC/SaftyPLC Instance <-> Device 1/Term 1 (EK1200)/Term 14 (EL2809)
//     PlcTask Outputs/GVL_Safety.HWSafetyOk <-> Channel 14/Output
//     PlcTask Outputs/GVL_Safety.HWerror <-> Channel 15/Output
//   SaftyPLC/SaftyPLC Instance <-> Device 1/Term 1 (EK1200)/Term 4 (EL1809)
//     PlcTask Inputs/GVL_Safety.HWReset <-> Channel 16/Input
//     PlcTask Inputs/GVL_Safety.HWStart <-> Channel 14/Input
//     PlcTask Inputs/GVL_Safety.HWStop <-> Channel 15/Input
//   SaftyPLC/SaftyPLC Instance <-> Device 1/Term 1 (EK1200)/Term 91 (EL2912)
//     PlcTask Inputs/GVL_Safety.SaeftyOk <-> StandardInputs/Standard Out Var 139
//     PlcTask Inputs/GVL_Safety.SafetyInRun <-> StandardInputs/Standard Out Var 73
//     PlcTask Outputs/GVL_Safety.Reset <-> StandardOutputs/Standard In Var 1
//     PlcTask Outputs/GVL_Safety.Run <-> StandardOutputs/Standard In Var 2
//     PlcTask Outputs/GVL_Safety.Start <-> StandardOutputs/Standard In Var 75
//   SaftyPLC/SaftyPLC Instance <-> Device 3 (EtherCAT Automation Protocol)/Box 28 (Publisher)
//     PlcTask Outputs/GVL_Safety.Reset <-> Command/Outputs/VarData/Reset
//     PlcTask Outputs/GVL_Safety.Run <-> Command/Outputs/VarData/Run
//   SaftyPLC/SaftyPLC Instance <-> Device 4 (EtherCAT)/Box 50 (AT5100-0100)
//     PlcTask Outputs/GVL_Safety.Reset <-> Module 1 (SAFETY)/SAFETY Standard Outputdata/Standard In Var 1
//     PlcTask Outputs/GVL_Safety.Run <-> Module 1 (SAFETY)/SAFETY Standard Outputdata/Standard In Var 2
//   SaftyPLC/SaftyPLC Instance <-> Device 4 (EtherCAT)/Box 51 (AT5100-0100)
//     PlcTask Outputs/GVL_Safety.Reset <-> Module 1 (SAFETY)/SAFETY Standard Outputdata/Standard In Var 1
//     PlcTask Outputs/GVL_Safety.Run <-> Module 1 (SAFETY)/SAFETY Standard Outputdata/Standard In Var 2
//   SaftyPLC/SaftyPLC Instance <-> Device 4 (EtherCAT)/Box 52 (AT5100-0100)
//     PlcTask Outputs/GVL_Safety.Reset <-> Module 1 (SAFETY)/SAFETY Standard Outputdata/Standard In Var 1
//     PlcTask Outputs/GVL_Safety.Run <-> Module 1 (SAFETY)/SAFETY Standard Outputdata/Standard In Var 2
//   SaftyPLC/SaftyPLC Instance <-> Device 4 (EtherCAT)/Box 53 (AT5100-0100)
//     PlcTask Outputs/GVL_Safety.Reset <-> Module 1 (SAFETY)/SAFETY Standard Outputdata/Standard In Var 1
//     PlcTask Outputs/GVL_Safety.Run <-> Module 1 (SAFETY)/SAFETY Standard Outputdata/Standard In Var 2
//   SaftyPLC/SaftyPLC Instance <-> Device 4 (EtherCAT)/Box 54 (AT5100-0100)
//     PlcTask Outputs/GVL_Safety.Reset <-> Module 1 (SAFETY)/SAFETY Standard Outputdata/Standard In Var 1
//     PlcTask Outputs/GVL_Safety.Run <-> Module 1 (SAFETY)/SAFETY Standard Outputdata/Standard In Var 2
//   SaftyPLC/SaftyPLC Instance <-> Device 4 (EtherCAT)/Box 55 (AT5100-0100)
//     PlcTask Outputs/GVL_Safety.Reset <-> Module 1 (SAFETY)/SAFETY Standard Outputdata/Standard In Var 1
//     PlcTask Outputs/GVL_Safety.Run <-> Module 1 (SAFETY)/SAFETY Standard Outputdata/Standard In Var 2
//   SaftyPLC/SaftyPLC Instance <-> Device 4 (EtherCAT)/Box 56 (AT5100-0100)
//     PlcTask Outputs/GVL_Safety.Reset <-> Module 1 (SAFETY)/SAFETY Standard Outputdata/Standard In Var 1
//     PlcTask Outputs/GVL_Safety.Run <-> Module 1 (SAFETY)/SAFETY Standard Outputdata/Standard In Var 2
//   SaftyPLC/SaftyPLC Instance <-> Device 4 (EtherCAT)/Box 57 (AT5100-0100)
//     PlcTask Outputs/GVL_Safety.Reset <-> Module 1 (SAFETY)/SAFETY Standard Outputdata/Standard In Var 1
//     PlcTask Outputs/GVL_Safety.Run <-> Module 1 (SAFETY)/SAFETY Standard Outputdata/Standard In Var 2
//   SaftyPLC/SaftyPLC Instance <-> Device 4 (EtherCAT)/Box 58 (AT5100-0100)
//     PlcTask Outputs/GVL_Safety.Reset <-> Module 1 (SAFETY)/SAFETY Standard Outputdata/Standard In Var 1
//     PlcTask Outputs/GVL_Safety.Run <-> Module 1 (SAFETY)/SAFETY Standard Outputdata/Standard In Var 2
//   SaftyPLC/SaftyPLC Instance <-> Device 4 (EtherCAT)/Box 59 (AT5100-0100)
//     PlcTask Outputs/GVL_Safety.Reset <-> Module 1 (SAFETY)/SAFETY Standard Outputdata/Standard In Var 1
//     PlcTask Outputs/GVL_Safety.Run <-> Module 1 (SAFETY)/SAFETY Standard Outputdata/Standard In Var 2
//   SaftyPLC/SaftyPLC Instance <-> Device 4 (EtherCAT)/Box 60 (AT5100-0100)
//     PlcTask Outputs/GVL_Safety.Reset <-> Module 1 (SAFETY)/SAFETY Standard Outputdata/Standard In Var 1
//     PlcTask Outputs/GVL_Safety.Run <-> Module 1 (SAFETY)/SAFETY Standard Outputdata/Standard In Var 2
//   SaftyPLC/SaftyPLC Instance <-> Device 4 (EtherCAT)/Box 61 (AT5100-0100)
//     PlcTask Outputs/GVL_Safety.Reset <-> Module 1 (SAFETY)/SAFETY Standard Outputdata/Standard In Var 1
//     PlcTask Outputs/GVL_Safety.Run <-> Module 1 (SAFETY)/SAFETY Standard Outputdata/Standard In Var 2
//   SaftyPLC/SaftyPLC Instance <-> Device 4 (EtherCAT)/Box 62 (AT5100-0100)
//     PlcTask Outputs/GVL_Safety.Reset <-> Module 1 (SAFETY)/SAFETY Standard Outputdata/Standard In Var 1
//     PlcTask Outputs/GVL_Safety.Run <-> Module 1 (SAFETY)/SAFETY Standard Outputdata/Standard In Var 2
//   SaftyPLC/SaftyPLC Instance <-> Device 4 (EtherCAT)/Box 63 (AT5100-0100)
//     PlcTask Outputs/GVL_Safety.Reset <-> Module 1 (SAFETY)/SAFETY Standard Outputdata/Standard In Var 1
//     PlcTask Outputs/GVL_Safety.Run <-> Module 1 (SAFETY)/SAFETY Standard Outputdata/Standard In Var 2
//   SaftyPLC/SaftyPLC Instance <-> Device 4 (EtherCAT)/Box 64 (AT5100-0100)
//     PlcTask Outputs/GVL_Safety.Reset <-> Module 1 (SAFETY)/SAFETY Standard Outputdata/Standard In Var 1
//     PlcTask Outputs/GVL_Safety.Run <-> Module 1 (SAFETY)/SAFETY Standard Outputdata/Standard In Var 2
//   SaftyPLC/SaftyPLC Instance <-> Device 4 (EtherCAT)/Box 65 (AT5100-0100)
//     PlcTask Outputs/GVL_Safety.Reset <-> Module 1 (SAFETY)/SAFETY Standard Outputdata/Standard In Var 1
//     PlcTask Outputs/GVL_Safety.Run <-> Module 1 (SAFETY)/SAFETY Standard Outputdata/Standard In Var 2
//   SaftyPLC/SaftyPLC Instance <-> Device 4 (EtherCAT)/Box 66 (AT5100-0100)
//     PlcTask Outputs/GVL_Safety.Reset <-> Module 1 (SAFETY)/SAFETY Standard Outputdata/Standard In Var 1
//     PlcTask Outputs/GVL_Safety.Run <-> Module 1 (SAFETY)/SAFETY Standard Outputdata/Standard In Var 2
//   SaftyPLC/SaftyPLC Instance <-> Device 4 (EtherCAT)/Box 67 (AT5100-0100)
//     PlcTask Outputs/GVL_Safety.Reset <-> Module 1 (SAFETY)/SAFETY Standard Outputdata/Standard In Var 1
//     PlcTask Outputs/GVL_Safety.Run <-> Module 1 (SAFETY)/SAFETY Standard Outputdata/Standard In Var 2
//   SaftyPLC/SaftyPLC Instance <-> Device 4 (EtherCAT)/Box 68 (AT5100-0100)
//     PlcTask Outputs/GVL_Safety.Reset <-> Module 1 (SAFETY)/SAFETY Standard Outputdata/Standard In Var 1
//     PlcTask Outputs/GVL_Safety.Run <-> Module 1 (SAFETY)/SAFETY Standard Outputdata/Standard In Var 2
//   SaftyPLC/SaftyPLC Instance <-> Device 4 (EtherCAT)/Box 69 (AT5100-0100)
//     PlcTask Outputs/GVL_Safety.Reset <-> Module 1 (SAFETY)/SAFETY Standard Outputdata/Standard In Var 1
//     PlcTask Outputs/GVL_Safety.Run <-> Module 1 (SAFETY)/SAFETY Standard Outputdata/Standard In Var 2
//   SaftyPLC/SaftyPLC Instance <-> Device 4 (EtherCAT)/Box 70 (AT5100-0100)
//     PlcTask Outputs/GVL_Safety.Reset <-> Module 1 (SAFETY)/SAFETY Standard Outputdata/Standard In Var 1
//     PlcTask Outputs/GVL_Safety.Run <-> Module 1 (SAFETY)/SAFETY Standard Outputdata/Standard In Var 2
//   SaftyPLC/SaftyPLC Instance <-> Device 4 (EtherCAT)/Box 71 (AT5100-0100)
//     PlcTask Outputs/GVL_Safety.Reset <-> Module 1 (SAFETY)/SAFETY Standard Outputdata/Standard In Var 1
//     PlcTask Outputs/GVL_Safety.Run <-> Module 1 (SAFETY)/SAFETY Standard Outputdata/Standard In Var 2
//   SaftyPLC/SaftyPLC Instance <-> Device 4 (EtherCAT)/Box 72 (AT5100-0100)
//     PlcTask Outputs/GVL_Safety.Reset <-> Module 1 (SAFETY)/SAFETY Standard Outputdata/Standard In Var 1
//     PlcTask Outputs/GVL_Safety.Run <-> Module 1 (SAFETY)/SAFETY Standard Outputdata/Standard In Var 2
//   SaftyPLC/SaftyPLC Instance <-> Device 4 (EtherCAT)/Box 73 (AT5100-0100)
//     PlcTask Outputs/GVL_Safety.Reset <-> Module 1 (SAFETY)/SAFETY Standard Outputdata/Standard In Var 1
//     PlcTask Outputs/GVL_Safety.Run <-> Module 1 (SAFETY)/SAFETY Standard Outputdata/Standard In Var 2
//   SaftyPLC/SaftyPLC Instance <-> Device 4 (EtherCAT)/Box 74 (AT5100-0100)
//     PlcTask Outputs/GVL_Safety.Reset <-> Module 1 (SAFETY)/SAFETY Standard Outputdata/Standard In Var 1
//     PlcTask Outputs/GVL_Safety.Run <-> Module 1 (SAFETY)/SAFETY Standard Outputdata/Standard In Var 2
//   SaftyPLC/SaftyPLC Instance <-> Device 4 (EtherCAT)/Box 75 (AT5100-0100)
//     PlcTask Outputs/GVL_Safety.Reset <-> Module 1 (SAFETY)/SAFETY Standard Outputdata/Standard In Var 1
//     PlcTask Outputs/GVL_Safety.Run <-> Module 1 (SAFETY)/SAFETY Standard Outputdata/Standard In Var 2
//   SaftyPLC/SaftyPLC Instance <-> Device 4 (EtherCAT)/Box 76 (AT5100-0100)
//     PlcTask Outputs/GVL_Safety.Reset <-> Module 1 (SAFETY)/SAFETY Standard Outputdata/Standard In Var 1
//     PlcTask Outputs/GVL_Safety.Run <-> Module 1 (SAFETY)/SAFETY Standard Outputdata/Standard In Var 2
//   SaftyPLC/SaftyPLC Instance <-> Device 5 (EtherCAT)/Box 1 (AT5840-0000)
//     PlcTask Outputs/GVL_IO.PowerSupplyReset <-> PSU Outputs/Reset
//   SaftyPLC/SaftyPLC Instance <-> Device 8 (EtherCAT)/Box 23 (AT5100-0100)
//     PlcTask Outputs/GVL_Safety.Reset <-> Module 1 (SAFETY)/SAFETY Standard Outputdata/Standard In Var 1
//     PlcTask Outputs/GVL_Safety.Run <-> Module 1 (SAFETY)/SAFETY Standard Outputdata/Standard In Var 2
//   SaftyPLC/SaftyPLC Instance <-> Device 8 (EtherCAT)/Box 24 (AT5100-0100)
//     PlcTask Outputs/GVL_Safety.Reset <-> Module 1 (SAFETY)/SAFETY Standard Outputdata/Standard In Var 1
//     PlcTask Outputs/GVL_Safety.Run <-> Module 1 (SAFETY)/SAFETY Standard Outputdata/Standard In Var 2
//   SaftyPLC/SaftyPLC Instance <-> Device 8 (EtherCAT)/Box 25 (AT5100-0100)
//     PlcTask Outputs/GVL_Safety.Reset <-> Module 1 (SAFETY)/SAFETY Standard Outputdata/Standard In Var 1
//     PlcTask Outputs/GVL_Safety.Run <-> Module 1 (SAFETY)/SAFETY Standard Outputdata/Standard In Var 2
//   SaftyPLC/SaftyPLC Instance <-> Device 8 (EtherCAT)/Box 26 (AT5100-0100)
//     PlcTask Outputs/GVL_Safety.Reset <-> Module 1 (SAFETY)/SAFETY Standard Outputdata/Standard In Var 1
//     PlcTask Outputs/GVL_Safety.Run <-> Module 1 (SAFETY)/SAFETY Standard Outputdata/Standard In Var 2
//   SaftyPLC/SaftyPLC Instance <-> Device 8 (EtherCAT)/Box 27 (AT5100-0100)
//     PlcTask Outputs/GVL_Safety.Reset <-> Module 1 (SAFETY)/SAFETY Standard Outputdata/Standard In Var 1
//     PlcTask Outputs/GVL_Safety.Run <-> Module 1 (SAFETY)/SAFETY Standard Outputdata/Standard In Var 2
//   SaftyPLC/SaftyPLC Instance <-> Device 8 (EtherCAT)/Box 28 (AT5100-0100)
//     PlcTask Outputs/GVL_Safety.Reset <-> Module 1 (SAFETY)/SAFETY Standard Outputdata/Standard In Var 1
//     PlcTask Outputs/GVL_Safety.Run <-> Module 1 (SAFETY)/SAFETY Standard Outputdata/Standard In Var 2
//   SaftyPLC/SaftyPLC Instance <-> Device 8 (EtherCAT)/Box 29 (AT5100-0100)
//     PlcTask Outputs/GVL_Safety.Reset <-> Module 1 (SAFETY)/SAFETY Standard Outputdata/Standard In Var 1
//     PlcTask Outputs/GVL_Safety.Run <-> Module 1 (SAFETY)/SAFETY Standard Outputdata/Standard In Var 2
//   SaftyPLC/SaftyPLC Instance <-> Device 8 (EtherCAT)/Box 30 (AT5100-0100)
//     PlcTask Outputs/GVL_Safety.Reset <-> Module 1 (SAFETY)/SAFETY Standard Outputdata/Standard In Var 1
//     PlcTask Outputs/GVL_Safety.Run <-> Module 1 (SAFETY)/SAFETY Standard Outputdata/Standard In Var 2
//   SaftyPLC/SaftyPLC Instance <-> Device 8 (EtherCAT)/Box 31 (AT5100-0100)
//     PlcTask Outputs/GVL_Safety.Reset <-> Module 1 (SAFETY)/SAFETY Standard Outputdata/Standard In Var 1
//     PlcTask Outputs/GVL_Safety.Run <-> Module 1 (SAFETY)/SAFETY Standard Outputdata/Standard In Var 2
//   SaftyPLC/SaftyPLC Instance <-> Device 8 (EtherCAT)/Box 32 (AT5100-0100)
//     PlcTask Outputs/GVL_Safety.Reset <-> Module 1 (SAFETY)/SAFETY Standard Outputdata/Standard In Var 1
//     PlcTask Outputs/GVL_Safety.Run <-> Module 1 (SAFETY)/SAFETY Standard Outputdata/Standard In Var 2
//   SaftyPLC/SaftyPLC Instance <-> Device 8 (EtherCAT)/Box 33 (AT5100-0100)
//     PlcTask Outputs/GVL_Safety.Reset <-> Module 1 (SAFETY)/SAFETY Standard Outputdata/Standard In Var 1
//     PlcTask Outputs/GVL_Safety.Run <-> Module 1 (SAFETY)/SAFETY Standard Outputdata/Standard In Var 2
//   SaftyPLC/SaftyPLC Instance <-> Device 8 (EtherCAT)/Box 34 (AT5100-0100)
//     PlcTask Outputs/GVL_Safety.Reset <-> Module 1 (SAFETY)/SAFETY Standard Outputdata/Standard In Var 1
//     PlcTask Outputs/GVL_Safety.Run <-> Module 1 (SAFETY)/SAFETY Standard Outputdata/Standard In Var 2
//   SaftyPLC/SaftyPLC Instance <-> Device 8 (EtherCAT)/Box 35 (AT5100-0100)
//     PlcTask Outputs/GVL_Safety.Reset <-> Module 1 (SAFETY)/SAFETY Standard Outputdata/Standard In Var 1
//     PlcTask Outputs/GVL_Safety.Run <-> Module 1 (SAFETY)/SAFETY Standard Outputdata/Standard In Var 2
//   SaftyPLC/SaftyPLC Instance <-> Device 8 (EtherCAT)/Box 36 (AT5100-0100)
//     PlcTask Outputs/GVL_Safety.Reset <-> Module 1 (SAFETY)/SAFETY Standard Outputdata/Standard In Var 1
//     PlcTask Outputs/GVL_Safety.Run <-> Module 1 (SAFETY)/SAFETY Standard Outputdata/Standard In Var 2
//   SaftyPLC/SaftyPLC Instance <-> Device 8 (EtherCAT)/Box 37 (AT5100-0100)
//     PlcTask Outputs/GVL_Safety.Reset <-> Module 1 (SAFETY)/SAFETY Standard Outputdata/Standard In Var 1
//     PlcTask Outputs/GVL_Safety.Run <-> Module 1 (SAFETY)/SAFETY Standard Outputdata/Standard In Var 2
//   SaftyPLC/SaftyPLC Instance <-> Device 8 (EtherCAT)/Box 38 (AT5100-0100)
//     PlcTask Outputs/GVL_Safety.Reset <-> Module 1 (SAFETY)/SAFETY Standard Outputdata/Standard In Var 1
//     PlcTask Outputs/GVL_Safety.Run <-> Module 1 (SAFETY)/SAFETY Standard Outputdata/Standard In Var 2
//   SaftyPLC/SaftyPLC Instance <-> Device 8 (EtherCAT)/Box 39 (AT5100-0100)
//     PlcTask Outputs/GVL_Safety.Reset <-> Module 1 (SAFETY)/SAFETY Standard Outputdata/Standard In Var 1
//     PlcTask Outputs/GVL_Safety.Run <-> Module 1 (SAFETY)/SAFETY Standard Outputdata/Standard In Var 2
//   SaftyPLC/SaftyPLC Instance <-> Device 8 (EtherCAT)/Box 40 (AT5100-0100)
//     PlcTask Outputs/GVL_Safety.Reset <-> Module 1 (SAFETY)/SAFETY Standard Outputdata/Standard In Var 1
//     PlcTask Outputs/GVL_Safety.Run <-> Module 1 (SAFETY)/SAFETY Standard Outputdata/Standard In Var 2
//   SaftyPLC/SaftyPLC Instance <-> Device 8 (EtherCAT)/Box 41 (AT5100-0100)
//     PlcTask Outputs/GVL_Safety.Reset <-> Module 1 (SAFETY)/SAFETY Standard Outputdata/Standard In Var 1
//     PlcTask Outputs/GVL_Safety.Run <-> Module 1 (SAFETY)/SAFETY Standard Outputdata/Standard In Var 2
//   SaftyPLC/SaftyPLC Instance <-> Device 8 (EtherCAT)/Box 42 (AT5100-0100)
//     PlcTask Outputs/GVL_Safety.Reset <-> Module 1 (SAFETY)/SAFETY Standard Outputdata/Standard In Var 1
//     PlcTask Outputs/GVL_Safety.Run <-> Module 1 (SAFETY)/SAFETY Standard Outputdata/Standard In Var 2
//   SaftyPLC/SaftyPLC Instance <-> Device 8 (EtherCAT)/Box 43 (AT5100-0100)
//     PlcTask Outputs/GVL_Safety.Reset <-> Module 1 (SAFETY)/SAFETY Standard Outputdata/Standard In Var 1
//     PlcTask Outputs/GVL_Safety.Run <-> Module 1 (SAFETY)/SAFETY Standard Outputdata/Standard In Var 2
//   SaftyPLC/SaftyPLC Instance <-> Device 8 (EtherCAT)/Box 44 (AT5100-0100)
//     PlcTask Outputs/GVL_Safety.Reset <-> Module 1 (SAFETY)/SAFETY Standard Outputdata/Standard In Var 1
//     PlcTask Outputs/GVL_Safety.Run <-> Module 1 (SAFETY)/SAFETY Standard Outputdata/Standard In Var 2
//   SaftyPLC/SaftyPLC Instance <-> Device 8 (EtherCAT)/Box 45 (AT5100-0100)
//     PlcTask Outputs/GVL_Safety.Reset <-> Module 1 (SAFETY)/SAFETY Standard Outputdata/Standard In Var 1
//     PlcTask Outputs/GVL_Safety.Run <-> Module 1 (SAFETY)/SAFETY Standard Outputdata/Standard In Var 2
//   SaftyPLC/SaftyPLC Instance <-> Device 8 (EtherCAT)/Box 46 (AT5100-0100)
//     PlcTask Outputs/GVL_Safety.Reset <-> Module 1 (SAFETY)/SAFETY Standard Outputdata/Standard In Var 1
//     PlcTask Outputs/GVL_Safety.Run <-> Module 1 (SAFETY)/SAFETY Standard Outputdata/Standard In Var 2
//   SaftyPLC/SaftyPLC Instance <-> Device 8 (EtherCAT)/Box 47 (AT5100-0100)
//     PlcTask Outputs/GVL_Safety.Reset <-> Module 1 (SAFETY)/SAFETY Standard Outputdata/Standard In Var 1
//     PlcTask Outputs/GVL_Safety.Run <-> Module 1 (SAFETY)/SAFETY Standard Outputdata/Standard In Var 2
//   SaftyPLC/SaftyPLC Instance <-> Device 8 (EtherCAT)/Box 48 (AT5100-0100)
//     PlcTask Outputs/GVL_Safety.Reset <-> Module 1 (SAFETY)/SAFETY Standard Outputdata/Standard In Var 1
//     PlcTask Outputs/GVL_Safety.Run <-> Module 1 (SAFETY)/SAFETY Standard Outputdata/Standard In Var 2
//   SaftyPLC/SaftyPLC Instance <-> Device 8 (EtherCAT)/Box 49 (AT5100-0100)
//     PlcTask Outputs/GVL_Safety.Reset <-> Module 1 (SAFETY)/SAFETY Standard Outputdata/Standard In Var 1
//     PlcTask Outputs/GVL_Safety.Run <-> Module 1 (SAFETY)/SAFETY Standard Outputdata/Standard In Var 2
//   (this object) <-> TcCOM Objects/XTS ProcessingUnit 1/XL Part 1/XL Module 19
//     Box 38 (AT5100-0100)/DRV Commutation angle/Commutation angle <-> Data Pointer/CommutationAngle
//     Box 38 (AT5100-0100)/DRV Controlword/Controlword <-> Data Pointer/Control
//     Box 38 (AT5100-0100)/DRV Statusword/Statusword <-> Data Pointer/Status
//     Box 38 (AT5100-0100)/DRV Target torque/Target torque <-> Data Pointer/Torque
//     Box 38 (AT5100-0100)/DRV Torque actual value/Torque actual value <-> Data Pointer/ActTorque
//     Box 38 (AT5100-0100)/XFB Inputs/Data <-> Data Pointer/HallSensorValues
//   (this object) <-> TcCOM Objects/XTS ProcessingUnit 1/XL Part 1/XL Module 20
//     Box 39 (AT5100-0100)/DRV Commutation angle/Commutation angle <-> Data Pointer/CommutationAngle
//     Box 39 (AT5100-0100)/DRV Controlword/Controlword <-> Data Pointer/Control
//     Box 39 (AT5100-0100)/DRV Statusword/Statusword <-> Data Pointer/Status
//     Box 39 (AT5100-0100)/DRV Target torque/Target torque <-> Data Pointer/Torque
//     Box 39 (AT5100-0100)/DRV Torque actual value/Torque actual value <-> Data Pointer/ActTorque
//     Box 39 (AT5100-0100)/XFB Inputs/Data <-> Data Pointer/HallSensorValues
//   (this object) <-> TcCOM Objects/XTS ProcessingUnit 1/XL Part 1/XL Module 21
//     Box 40 (AT5100-0100)/DRV Commutation angle/Commutation angle <-> Data Pointer/CommutationAngle
//     Box 40 (AT5100-0100)/DRV Controlword/Controlword <-> Data Pointer/Control
//     Box 40 (AT5100-0100)/DRV Statusword/Statusword <-> Data Pointer/Status
//     Box 40 (AT5100-0100)/DRV Target torque/Target torque <-> Data Pointer/Torque
//     Box 40 (AT5100-0100)/DRV Torque actual value/Torque actual value <-> Data Pointer/ActTorque
//     Box 40 (AT5100-0100)/XFB Inputs/Data <-> Data Pointer/HallSensorValues
//   (this object) <-> TcCOM Objects/XTS ProcessingUnit 1/XL Part 1/XL Module 22
//     Box 41 (AT5100-0100)/DRV Commutation angle/Commutation angle <-> Data Pointer/CommutationAngle
//     Box 41 (AT5100-0100)/DRV Controlword/Controlword <-> Data Pointer/Control
//     Box 41 (AT5100-0100)/DRV Statusword/Statusword <-> Data Pointer/Status
//     Box 41 (AT5100-0100)/DRV Target torque/Target torque <-> Data Pointer/Torque
//     Box 41 (AT5100-0100)/DRV Torque actual value/Torque actual value <-> Data Pointer/ActTorque
//     Box 41 (AT5100-0100)/XFB Inputs/Data <-> Data Pointer/HallSensorValues
//   (this object) <-> TcCOM Objects/XTS ProcessingUnit 1/XL Part 1/XL Module 26
//     Box 42 (AT5100-0100)/DRV Commutation angle/Commutation angle <-> Data Pointer/CommutationAngle
//     Box 42 (AT5100-0100)/DRV Controlword/Controlword <-> Data Pointer/Control
//     Box 42 (AT5100-0100)/DRV Statusword/Statusword <-> Data Pointer/Status
//     Box 42 (AT5100-0100)/DRV Target torque/Target torque <-> Data Pointer/Torque
//     Box 42 (AT5100-0100)/DRV Torque actual value/Torque actual value <-> Data Pointer/ActTorque
//     Box 42 (AT5100-0100)/XFB Inputs/Data <-> Data Pointer/HallSensorValues
//   (this object) <-> TcCOM Objects/XTS ProcessingUnit 1/XL Part 1/XL Module 27
//     Box 43 (AT5100-0100)/DRV Commutation angle/Commutation angle <-> Data Pointer/CommutationAngle
//     Box 43 (AT5100-0100)/DRV Controlword/Controlword <-> Data Pointer/Control
//     Box 43 (AT5100-0100)/DRV Statusword/Statusword <-> Data Pointer/Status
//     Box 43 (AT5100-0100)/DRV Target torque/Target torque <-> Data Pointer/Torque
//     Box 43 (AT5100-0100)/DRV Torque actual value/Torque actual value <-> Data Pointer/ActTorque
//     Box 43 (AT5100-0100)/XFB Inputs/Data <-> Data Pointer/HallSensorValues
//   (this object) <-> TcCOM Objects/XTS ProcessingUnit 1/XL Part 1/XL Module 28
//     Box 44 (AT5100-0100)/DRV Commutation angle/Commutation angle <-> Data Pointer/CommutationAngle
//     Box 44 (AT5100-0100)/DRV Controlword/Controlword <-> Data Pointer/Control
//     Box 44 (AT5100-0100)/DRV Statusword/Statusword <-> Data Pointer/Status
//     Box 44 (AT5100-0100)/DRV Target torque/Target torque <-> Data Pointer/Torque
//     Box 44 (AT5100-0100)/DRV Torque actual value/Torque actual value <-> Data Pointer/ActTorque
//     Box 44 (AT5100-0100)/XFB Inputs/Data <-> Data Pointer/HallSensorValues
//   (this object) <-> TcCOM Objects/XTS ProcessingUnit 1/XL Part 1/XL Module 29
//     Box 45 (AT5100-0100)/DRV Commutation angle/Commutation angle <-> Data Pointer/CommutationAngle
//     Box 45 (AT5100-0100)/DRV Controlword/Controlword <-> Data Pointer/Control
//     Box 45 (AT5100-0100)/DRV Statusword/Statusword <-> Data Pointer/Status
//     Box 45 (AT5100-0100)/DRV Target torque/Target torque <-> Data Pointer/Torque
//     Box 45 (AT5100-0100)/DRV Torque actual value/Torque actual value <-> Data Pointer/ActTorque
//     Box 45 (AT5100-0100)/XFB Inputs/Data <-> Data Pointer/HallSensorValues
//   (this object) <-> TcCOM Objects/XTS ProcessingUnit 1/XL Part 1/XL Module 30
//     Box 46 (AT5100-0100)/DRV Commutation angle/Commutation angle <-> Data Pointer/CommutationAngle
//     Box 46 (AT5100-0100)/DRV Controlword/Controlword <-> Data Pointer/Control
//     Box 46 (AT5100-0100)/DRV Statusword/Statusword <-> Data Pointer/Status
//     Box 46 (AT5100-0100)/DRV Target torque/Target torque <-> Data Pointer/Torque
//     Box 46 (AT5100-0100)/DRV Torque actual value/Torque actual value <-> Data Pointer/ActTorque
//     Box 46 (AT5100-0100)/XFB Inputs/Data <-> Data Pointer/HallSensorValues
//   (this object) <-> TcCOM Objects/XTS ProcessingUnit 1/XL Part 1/XL Module 31
//     Box 47 (AT5100-0100)/DRV Commutation angle/Commutation angle <-> Data Pointer/CommutationAngle
//     Box 47 (AT5100-0100)/DRV Controlword/Controlword <-> Data Pointer/Control
//     Box 47 (AT5100-0100)/DRV Statusword/Statusword <-> Data Pointer/Status
//     Box 47 (AT5100-0100)/DRV Target torque/Target torque <-> Data Pointer/Torque
//     Box 47 (AT5100-0100)/DRV Torque actual value/Torque actual value <-> Data Pointer/ActTorque
//     Box 47 (AT5100-0100)/XFB Inputs/Data <-> Data Pointer/HallSensorValues
//   (this object) <-> TcCOM Objects/XTS ProcessingUnit 1/XL Part 1/XL Module 32
//     Box 48 (AT5100-0100)/DRV Commutation angle/Commutation angle <-> Data Pointer/CommutationAngle
//     Box 48 (AT5100-0100)/DRV Controlword/Controlword <-> Data Pointer/Control
//     Box 48 (AT5100-0100)/DRV Statusword/Statusword <-> Data Pointer/Status
//     Box 48 (AT5100-0100)/DRV Target torque/Target torque <-> Data Pointer/Torque
//     Box 48 (AT5100-0100)/DRV Torque actual value/Torque actual value <-> Data Pointer/ActTorque
//     Box 48 (AT5100-0100)/XFB Inputs/Data <-> Data Pointer/HallSensorValues
//   (this object) <-> TcCOM Objects/XTS ProcessingUnit 1/XL Part 1/XL Module 33
//     Box 49 (AT5100-0100)/DRV Commutation angle/Commutation angle <-> Data Pointer/CommutationAngle
//     Box 49 (AT5100-0100)/DRV Controlword/Controlword <-> Data Pointer/Control
//     Box 49 (AT5100-0100)/DRV Statusword/Statusword <-> Data Pointer/Status
//     Box 49 (AT5100-0100)/DRV Target torque/Target torque <-> Data Pointer/Torque
//     Box 49 (AT5100-0100)/DRV Torque actual value/Torque actual value <-> Data Pointer/ActTorque
//     Box 49 (AT5100-0100)/XFB Inputs/Data <-> Data Pointer/HallSensorValues
//   (this object) <-> TcCOM Objects/XTS ProcessingUnit 1/XL Part 2/XL Module 23
//     Box 37 (AT5100-0100)/DRV Commutation angle/Commutation angle <-> Data Pointer/CommutationAngle
//     Box 37 (AT5100-0100)/DRV Controlword/Controlword <-> Data Pointer/Control
//     Box 37 (AT5100-0100)/DRV Statusword/Statusword <-> Data Pointer/Status
//     Box 37 (AT5100-0100)/DRV Target torque/Target torque <-> Data Pointer/Torque
//     Box 37 (AT5100-0100)/DRV Torque actual value/Torque actual value <-> Data Pointer/ActTorque
//     Box 37 (AT5100-0100)/XFB Inputs/Data <-> Data Pointer/HallSensorValues
//   (this object) <-> TcCOM Objects/XTS ProcessingUnit 1/XL Part 2/XL Module 24
//     Box 28 (AT5100-0100)/DRV Commutation angle/Commutation angle <-> Data Pointer/CommutationAngle
//     Box 28 (AT5100-0100)/DRV Controlword/Controlword <-> Data Pointer/Control
//     Box 28 (AT5100-0100)/DRV Statusword/Statusword <-> Data Pointer/Status
//     Box 28 (AT5100-0100)/DRV Target torque/Target torque <-> Data Pointer/Torque
//     Box 28 (AT5100-0100)/DRV Torque actual value/Torque actual value <-> Data Pointer/ActTorque
//     Box 28 (AT5100-0100)/XFB Inputs/Data <-> Data Pointer/HallSensorValues
//   (this object) <-> TcCOM Objects/XTS ProcessingUnit 1/XL Part 2/XL Module 25
//     Box 29 (AT5100-0100)/DRV Commutation angle/Commutation angle <-> Data Pointer/CommutationAngle
//     Box 29 (AT5100-0100)/DRV Controlword/Controlword <-> Data Pointer/Control
//     Box 29 (AT5100-0100)/DRV Statusword/Statusword <-> Data Pointer/Status
//     Box 29 (AT5100-0100)/DRV Target torque/Target torque <-> Data Pointer/Torque
//     Box 29 (AT5100-0100)/DRV Torque actual value/Torque actual value <-> Data Pointer/ActTorque
//     Box 29 (AT5100-0100)/XFB Inputs/Data <-> Data Pointer/HallSensorValues
//   (this object) <-> TcCOM Objects/XTS ProcessingUnit 1/XL Part 2/XL Module 58
//     Box 30 (AT5100-0100)/DRV Commutation angle/Commutation angle <-> Data Pointer/CommutationAngle
//     Box 30 (AT5100-0100)/DRV Controlword/Controlword <-> Data Pointer/Control
//     Box 30 (AT5100-0100)/DRV Statusword/Statusword <-> Data Pointer/Status
//     Box 30 (AT5100-0100)/DRV Target torque/Target torque <-> Data Pointer/Torque
//     Box 30 (AT5100-0100)/DRV Torque actual value/Torque actual value <-> Data Pointer/ActTorque
//     Box 30 (AT5100-0100)/XFB Inputs/Data <-> Data Pointer/HallSensorValues
//   (this object) <-> TcCOM Objects/XTS ProcessingUnit 1/XL Part 2/XL Module 59
//     Box 31 (AT5100-0100)/DRV Commutation angle/Commutation angle <-> Data Pointer/CommutationAngle
//     Box 31 (AT5100-0100)/DRV Controlword/Controlword <-> Data Pointer/Control
//     Box 31 (AT5100-0100)/DRV Statusword/Statusword <-> Data Pointer/Status
//     Box 31 (AT5100-0100)/DRV Target torque/Target torque <-> Data Pointer/Torque
//     Box 31 (AT5100-0100)/DRV Torque actual value/Torque actual value <-> Data Pointer/ActTorque
//     Box 31 (AT5100-0100)/XFB Inputs/Data <-> Data Pointer/HallSensorValues
//   (this object) <-> TcCOM Objects/XTS ProcessingUnit 1/XL Part 2/XL Module 60
//     Box 32 (AT5100-0100)/DRV Commutation angle/Commutation angle <-> Data Pointer/CommutationAngle
//     Box 32 (AT5100-0100)/DRV Controlword/Controlword <-> Data Pointer/Control
//     Box 32 (AT5100-0100)/DRV Statusword/Statusword <-> Data Pointer/Status
//     Box 32 (AT5100-0100)/DRV Target torque/Target torque <-> Data Pointer/Torque
//     Box 32 (AT5100-0100)/DRV Torque actual value/Torque actual value <-> Data Pointer/ActTorque
//     Box 32 (AT5100-0100)/XFB Inputs/Data <-> Data Pointer/HallSensorValues
//   (this object) <-> TcCOM Objects/XTS ProcessingUnit 1/XL Part 2/XL Module 61
//     Box 33 (AT5100-0100)/DRV Commutation angle/Commutation angle <-> Data Pointer/CommutationAngle
//     Box 33 (AT5100-0100)/DRV Controlword/Controlword <-> Data Pointer/Control
//     Box 33 (AT5100-0100)/DRV Statusword/Statusword <-> Data Pointer/Status
//     Box 33 (AT5100-0100)/DRV Target torque/Target torque <-> Data Pointer/Torque
//     Box 33 (AT5100-0100)/DRV Torque actual value/Torque actual value <-> Data Pointer/ActTorque
//     Box 33 (AT5100-0100)/XFB Inputs/Data <-> Data Pointer/HallSensorValues
//   (this object) <-> TcCOM Objects/XTS ProcessingUnit 1/XL Part 2/XL Module 62
//     Box 34 (AT5100-0100)/DRV Commutation angle/Commutation angle <-> Data Pointer/CommutationAngle
//     Box 34 (AT5100-0100)/DRV Controlword/Controlword <-> Data Pointer/Control
//     Box 34 (AT5100-0100)/DRV Statusword/Statusword <-> Data Pointer/Status
//     Box 34 (AT5100-0100)/DRV Target torque/Target torque <-> Data Pointer/Torque
//     Box 34 (AT5100-0100)/DRV Torque actual value/Torque actual value <-> Data Pointer/ActTorque
//     Box 34 (AT5100-0100)/XFB Inputs/Data <-> Data Pointer/HallSensorValues
//   (this object) <-> TcCOM Objects/XTS ProcessingUnit 1/XL Part 2/XL Module 63
//     Box 35 (AT5100-0100)/DRV Commutation angle/Commutation angle <-> Data Pointer/CommutationAngle
//     Box 35 (AT5100-0100)/DRV Controlword/Controlword <-> Data Pointer/Control
//     Box 35 (AT5100-0100)/DRV Statusword/Statusword <-> Data Pointer/Status
//     Box 35 (AT5100-0100)/DRV Target torque/Target torque <-> Data Pointer/Torque
//     Box 35 (AT5100-0100)/DRV Torque actual value/Torque actual value <-> Data Pointer/ActTorque
//     Box 35 (AT5100-0100)/XFB Inputs/Data <-> Data Pointer/HallSensorValues
//   (this object) <-> TcCOM Objects/XTS ProcessingUnit 1/XL Part 2/XL Module 64
//     Box 36 (AT5100-0100)/DRV Commutation angle/Commutation angle <-> Data Pointer/CommutationAngle
//     Box 36 (AT5100-0100)/DRV Controlword/Controlword <-> Data Pointer/Control
//     Box 36 (AT5100-0100)/DRV Statusword/Statusword <-> Data Pointer/Status
//     Box 36 (AT5100-0100)/DRV Target torque/Target torque <-> Data Pointer/Torque
//     Box 36 (AT5100-0100)/DRV Torque actual value/Torque actual value <-> Data Pointer/ActTorque
//     Box 36 (AT5100-0100)/XFB Inputs/Data <-> Data Pointer/HallSensorValues
//   (this object) <-> TcCOM Objects/XTS ProcessingUnit 1/XL Part End/XL Module 14
//     Box 23 (AT5100-0100)/DRV Commutation angle/Commutation angle <-> Data Pointer/CommutationAngle
//     Box 23 (AT5100-0100)/DRV Controlword/Controlword <-> Data Pointer/Control
//     Box 23 (AT5100-0100)/DRV Statusword/Statusword <-> Data Pointer/Status
//     Box 23 (AT5100-0100)/DRV Target torque/Target torque <-> Data Pointer/Torque
//     Box 23 (AT5100-0100)/DRV Torque actual value/Torque actual value <-> Data Pointer/ActTorque
//     Box 23 (AT5100-0100)/XFB Inputs/Data <-> Data Pointer/HallSensorValues
//   (this object) <-> TcCOM Objects/XTS ProcessingUnit 1/XL Part End/XL Module 15
//     Box 24 (AT5100-0100)/DRV Commutation angle/Commutation angle <-> Data Pointer/CommutationAngle
//     Box 24 (AT5100-0100)/DRV Controlword/Controlword <-> Data Pointer/Control
//     Box 24 (AT5100-0100)/DRV Statusword/Statusword <-> Data Pointer/Status
//     Box 24 (AT5100-0100)/DRV Target torque/Target torque <-> Data Pointer/Torque
//     Box 24 (AT5100-0100)/DRV Torque actual value/Torque actual value <-> Data Pointer/ActTorque
//     Box 24 (AT5100-0100)/XFB Inputs/Data <-> Data Pointer/HallSensorValues
//   (this object) <-> TcCOM Objects/XTS ProcessingUnit 1/XL Part End/XL Module 16
//     Box 25 (AT5100-0100)/DRV Commutation angle/Commutation angle <-> Data Pointer/CommutationAngle
//     Box 25 (AT5100-0100)/DRV Controlword/Controlword <-> Data Pointer/Control
//     Box 25 (AT5100-0100)/DRV Statusword/Statusword <-> Data Pointer/Status
//     Box 25 (AT5100-0100)/DRV Target torque/Target torque <-> Data Pointer/Torque
//     Box 25 (AT5100-0100)/DRV Torque actual value/Torque actual value <-> Data Pointer/ActTorque
//     Box 25 (AT5100-0100)/XFB Inputs/Data <-> Data Pointer/HallSensorValues
//   (this object) <-> TcCOM Objects/XTS ProcessingUnit 1/XL Part End/XL Module 17
//     Box 26 (AT5100-0100)/DRV Commutation angle/Commutation angle <-> Data Pointer/CommutationAngle
//     Box 26 (AT5100-0100)/DRV Controlword/Controlword <-> Data Pointer/Control
//     Box 26 (AT5100-0100)/DRV Statusword/Statusword <-> Data Pointer/Status
//     Box 26 (AT5100-0100)/DRV Target torque/Target torque <-> Data Pointer/Torque
//     Box 26 (AT5100-0100)/DRV Torque actual value/Torque actual value <-> Data Pointer/ActTorque
//     Box 26 (AT5100-0100)/XFB Inputs/Data <-> Data Pointer/HallSensorValues
//   (this object) <-> TcCOM Objects/XTS ProcessingUnit 1/XL Part End/XL Module 18
//     Box 27 (AT5100-0100)/DRV Commutation angle/Commutation angle <-> Data Pointer/CommutationAngle
//     Box 27 (AT5100-0100)/DRV Controlword/Controlword <-> Data Pointer/Control
//     Box 27 (AT5100-0100)/DRV Statusword/Statusword <-> Data Pointer/Status
//     Box 27 (AT5100-0100)/DRV Target torque/Target torque <-> Data Pointer/Torque
//     Box 27 (AT5100-0100)/DRV Torque actual value/Torque actual value <-> Data Pointer/ActTorque
//     Box 27 (AT5100-0100)/XFB Inputs/Data <-> Data Pointer/HallSensorValues
//   (this object) <-> TcCOM Objects/XTS ProcessingUnit 1/XL Part 1/XL Module 34
//     Box 50 (AT5100-0100)/DRV Commutation angle/Commutation angle <-> Data Pointer/CommutationAngle
//     Box 50 (AT5100-0100)/DRV Controlword/Controlword <-> Data Pointer/Control
//     Box 50 (AT5100-0100)/DRV Statusword/Statusword <-> Data Pointer/Status
//     Box 50 (AT5100-0100)/DRV Target torque/Target torque <-> Data Pointer/Torque
//     Box 50 (AT5100-0100)/DRV Torque actual value/Torque actual value <-> Data Pointer/ActTorque
//     Box 50 (AT5100-0100)/XFB Inputs/Data <-> Data Pointer/HallSensorValues
//   (this object) <-> TcCOM Objects/XTS ProcessingUnit 1/XL Part 1/XL Module 35
//     Box 51 (AT5100-0100)/DRV Commutation angle/Commutation angle <-> Data Pointer/CommutationAngle
//     Box 51 (AT5100-0100)/DRV Controlword/Controlword <-> Data Pointer/Control
//     Box 51 (AT5100-0100)/DRV Statusword/Statusword <-> Data Pointer/Status
//     Box 51 (AT5100-0100)/DRV Target torque/Target torque <-> Data Pointer/Torque
//     Box 51 (AT5100-0100)/DRV Torque actual value/Torque actual value <-> Data Pointer/ActTorque
//     Box 51 (AT5100-0100)/XFB Inputs/Data <-> Data Pointer/HallSensorValues
//   (this object) <-> TcCOM Objects/XTS ProcessingUnit 1/XL Part 1/XL Module 36
//     Box 52 (AT5100-0100)/DRV Commutation angle/Commutation angle <-> Data Pointer/CommutationAngle
//     Box 52 (AT5100-0100)/DRV Controlword/Controlword <-> Data Pointer/Control
//     Box 52 (AT5100-0100)/DRV Statusword/Statusword <-> Data Pointer/Status
//     Box 52 (AT5100-0100)/DRV Target torque/Target torque <-> Data Pointer/Torque
//     Box 52 (AT5100-0100)/DRV Torque actual value/Torque actual value <-> Data Pointer/ActTorque
//     Box 52 (AT5100-0100)/XFB Inputs/Data <-> Data Pointer/HallSensorValues
//   (this object) <-> TcCOM Objects/XTS ProcessingUnit 1/XL Part 1/XL Module 37
//     Box 53 (AT5100-0100)/DRV Commutation angle/Commutation angle <-> Data Pointer/CommutationAngle
//     Box 53 (AT5100-0100)/DRV Controlword/Controlword <-> Data Pointer/Control
//     Box 53 (AT5100-0100)/DRV Statusword/Statusword <-> Data Pointer/Status
//     Box 53 (AT5100-0100)/DRV Target torque/Target torque <-> Data Pointer/Torque
//     Box 53 (AT5100-0100)/DRV Torque actual value/Torque actual value <-> Data Pointer/ActTorque
//     Box 53 (AT5100-0100)/XFB Inputs/Data <-> Data Pointer/HallSensorValues
//   (this object) <-> TcCOM Objects/XTS ProcessingUnit 1/XL Part 1/XL Module 38
//     Box 54 (AT5100-0100)/DRV Commutation angle/Commutation angle <-> Data Pointer/CommutationAngle
//     Box 54 (AT5100-0100)/DRV Controlword/Controlword <-> Data Pointer/Control
//     Box 54 (AT5100-0100)/DRV Statusword/Statusword <-> Data Pointer/Status
//     Box 54 (AT5100-0100)/DRV Target torque/Target torque <-> Data Pointer/Torque
//     Box 54 (AT5100-0100)/DRV Torque actual value/Torque actual value <-> Data Pointer/ActTorque
//     Box 54 (AT5100-0100)/XFB Inputs/Data <-> Data Pointer/HallSensorValues
//   (this object) <-> TcCOM Objects/XTS ProcessingUnit 1/XL Part 1/XL Module 39
//     Box 55 (AT5100-0100)/DRV Commutation angle/Commutation angle <-> Data Pointer/CommutationAngle
//     Box 55 (AT5100-0100)/DRV Controlword/Controlword <-> Data Pointer/Control
//     Box 55 (AT5100-0100)/DRV Statusword/Statusword <-> Data Pointer/Status
//     Box 55 (AT5100-0100)/DRV Target torque/Target torque <-> Data Pointer/Torque
//     Box 55 (AT5100-0100)/DRV Torque actual value/Torque actual value <-> Data Pointer/ActTorque
//     Box 55 (AT5100-0100)/XFB Inputs/Data <-> Data Pointer/HallSensorValues
//   (this object) <-> TcCOM Objects/XTS ProcessingUnit 1/XL Part 1/XL Module 40
//     Box 56 (AT5100-0100)/DRV Commutation angle/Commutation angle <-> Data Pointer/CommutationAngle
//     Box 56 (AT5100-0100)/DRV Controlword/Controlword <-> Data Pointer/Control
//     Box 56 (AT5100-0100)/DRV Statusword/Statusword <-> Data Pointer/Status
//     Box 56 (AT5100-0100)/DRV Target torque/Target torque <-> Data Pointer/Torque
//     Box 56 (AT5100-0100)/DRV Torque actual value/Torque actual value <-> Data Pointer/ActTorque
//     Box 56 (AT5100-0100)/XFB Inputs/Data <-> Data Pointer/HallSensorValues
//   (this object) <-> TcCOM Objects/XTS ProcessingUnit 1/XL Part 1/XL Module 41
//     Box 57 (AT5100-0100)/DRV Commutation angle/Commutation angle <-> Data Pointer/CommutationAngle
//     Box 57 (AT5100-0100)/DRV Controlword/Controlword <-> Data Pointer/Control
//     Box 57 (AT5100-0100)/DRV Statusword/Statusword <-> Data Pointer/Status
//     Box 57 (AT5100-0100)/DRV Target torque/Target torque <-> Data Pointer/Torque
//     Box 57 (AT5100-0100)/DRV Torque actual value/Torque actual value <-> Data Pointer/ActTorque
//     Box 57 (AT5100-0100)/XFB Inputs/Data <-> Data Pointer/HallSensorValues
//   (this object) <-> TcCOM Objects/XTS ProcessingUnit 1/XL Part 1/XL Module 42
//     Box 58 (AT5100-0100)/DRV Commutation angle/Commutation angle <-> Data Pointer/CommutationAngle
//     Box 58 (AT5100-0100)/DRV Controlword/Controlword <-> Data Pointer/Control
//     Box 58 (AT5100-0100)/DRV Statusword/Statusword <-> Data Pointer/Status
//     Box 58 (AT5100-0100)/DRV Target torque/Target torque <-> Data Pointer/Torque
//     Box 58 (AT5100-0100)/DRV Torque actual value/Torque actual value <-> Data Pointer/ActTorque
//     Box 58 (AT5100-0100)/XFB Inputs/Data <-> Data Pointer/HallSensorValues
//   (this object) <-> TcCOM Objects/XTS ProcessingUnit 1/XL Part 1/XL Module 43
//     Box 59 (AT5100-0100)/DRV Commutation angle/Commutation angle <-> Data Pointer/CommutationAngle
//     Box 59 (AT5100-0100)/DRV Controlword/Controlword <-> Data Pointer/Control
//     Box 59 (AT5100-0100)/DRV Statusword/Statusword <-> Data Pointer/Status
//     Box 59 (AT5100-0100)/DRV Target torque/Target torque <-> Data Pointer/Torque
//     Box 59 (AT5100-0100)/DRV Torque actual value/Torque actual value <-> Data Pointer/ActTorque
//     Box 59 (AT5100-0100)/XFB Inputs/Data <-> Data Pointer/HallSensorValues
//   (this object) <-> TcCOM Objects/XTS ProcessingUnit 1/XL Part 1/XL Module 44
//     Box 60 (AT5100-0100)/DRV Commutation angle/Commutation angle <-> Data Pointer/CommutationAngle
//     Box 60 (AT5100-0100)/DRV Controlword/Controlword <-> Data Pointer/Control
//     Box 60 (AT5100-0100)/DRV Statusword/Statusword <-> Data Pointer/Status
//     Box 60 (AT5100-0100)/DRV Target torque/Target torque <-> Data Pointer/Torque
//     Box 60 (AT5100-0100)/DRV Torque actual value/Torque actual value <-> Data Pointer/ActTorque
//     Box 60 (AT5100-0100)/XFB Inputs/Data <-> Data Pointer/HallSensorValues
//   (this object) <-> TcCOM Objects/XTS ProcessingUnit 1/XL Part 1/XL Module 45
//     Box 61 (AT5100-0100)/DRV Commutation angle/Commutation angle <-> Data Pointer/CommutationAngle
//     Box 61 (AT5100-0100)/DRV Controlword/Controlword <-> Data Pointer/Control
//     Box 61 (AT5100-0100)/DRV Statusword/Statusword <-> Data Pointer/Status
//     Box 61 (AT5100-0100)/DRV Target torque/Target torque <-> Data Pointer/Torque
//     Box 61 (AT5100-0100)/DRV Torque actual value/Torque actual value <-> Data Pointer/ActTorque
//     Box 61 (AT5100-0100)/XFB Inputs/Data <-> Data Pointer/HallSensorValues
//   (this object) <-> TcCOM Objects/XTS ProcessingUnit 1/XL Part 2/XL Module 48
//     Box 70 (AT5100-0100)/DRV Commutation angle/Commutation angle <-> Data Pointer/CommutationAngle
//     Box 70 (AT5100-0100)/DRV Controlword/Controlword <-> Data Pointer/Control
//     Box 70 (AT5100-0100)/DRV Statusword/Statusword <-> Data Pointer/Status
//     Box 70 (AT5100-0100)/DRV Target torque/Target torque <-> Data Pointer/Torque
//     Box 70 (AT5100-0100)/DRV Torque actual value/Torque actual value <-> Data Pointer/ActTorque
//     Box 70 (AT5100-0100)/XFB Inputs/Data <-> Data Pointer/HallSensorValues
//   (this object) <-> TcCOM Objects/XTS ProcessingUnit 1/XL Part 2/XL Module 49
//     Box 71 (AT5100-0100)/DRV Commutation angle/Commutation angle <-> Data Pointer/CommutationAngle
//     Box 71 (AT5100-0100)/DRV Controlword/Controlword <-> Data Pointer/Control
//     Box 71 (AT5100-0100)/DRV Statusword/Statusword <-> Data Pointer/Status
//     Box 71 (AT5100-0100)/DRV Target torque/Target torque <-> Data Pointer/Torque
//     Box 71 (AT5100-0100)/DRV Torque actual value/Torque actual value <-> Data Pointer/ActTorque
//     Box 71 (AT5100-0100)/XFB Inputs/Data <-> Data Pointer/HallSensorValues
//   (this object) <-> TcCOM Objects/XTS ProcessingUnit 1/XL Part 2/XL Module 50
//     Box 62 (AT5100-0100)/DRV Commutation angle/Commutation angle <-> Data Pointer/CommutationAngle
//     Box 62 (AT5100-0100)/DRV Controlword/Controlword <-> Data Pointer/Control
//     Box 62 (AT5100-0100)/DRV Statusword/Statusword <-> Data Pointer/Status
//     Box 62 (AT5100-0100)/DRV Target torque/Target torque <-> Data Pointer/Torque
//     Box 62 (AT5100-0100)/DRV Torque actual value/Torque actual value <-> Data Pointer/ActTorque
//     Box 62 (AT5100-0100)/XFB Inputs/Data <-> Data Pointer/HallSensorValues
//   (this object) <-> TcCOM Objects/XTS ProcessingUnit 1/XL Part 2/XL Module 51
//     Box 63 (AT5100-0100)/DRV Commutation angle/Commutation angle <-> Data Pointer/CommutationAngle
//     Box 63 (AT5100-0100)/DRV Controlword/Controlword <-> Data Pointer/Control
//     Box 63 (AT5100-0100)/DRV Statusword/Statusword <-> Data Pointer/Status
//     Box 63 (AT5100-0100)/DRV Target torque/Target torque <-> Data Pointer/Torque
//     Box 63 (AT5100-0100)/DRV Torque actual value/Torque actual value <-> Data Pointer/ActTorque
//     Box 63 (AT5100-0100)/XFB Inputs/Data <-> Data Pointer/HallSensorValues
//   (this object) <-> TcCOM Objects/XTS ProcessingUnit 1/XL Part 2/XL Module 52
//     Box 64 (AT5100-0100)/DRV Commutation angle/Commutation angle <-> Data Pointer/CommutationAngle
//     Box 64 (AT5100-0100)/DRV Controlword/Controlword <-> Data Pointer/Control
//     Box 64 (AT5100-0100)/DRV Statusword/Statusword <-> Data Pointer/Status
//     Box 64 (AT5100-0100)/DRV Target torque/Target torque <-> Data Pointer/Torque
//     Box 64 (AT5100-0100)/DRV Torque actual value/Torque actual value <-> Data Pointer/ActTorque
//     Box 64 (AT5100-0100)/XFB Inputs/Data <-> Data Pointer/HallSensorValues
//   (this object) <-> TcCOM Objects/XTS ProcessingUnit 1/XL Part 2/XL Module 53
//     Box 65 (AT5100-0100)/DRV Commutation angle/Commutation angle <-> Data Pointer/CommutationAngle
//     Box 65 (AT5100-0100)/DRV Controlword/Controlword <-> Data Pointer/Control
//     Box 65 (AT5100-0100)/DRV Statusword/Statusword <-> Data Pointer/Status
//     Box 65 (AT5100-0100)/DRV Target torque/Target torque <-> Data Pointer/Torque
//     Box 65 (AT5100-0100)/DRV Torque actual value/Torque actual value <-> Data Pointer/ActTorque
//     Box 65 (AT5100-0100)/XFB Inputs/Data <-> Data Pointer/HallSensorValues
//   (this object) <-> TcCOM Objects/XTS ProcessingUnit 1/XL Part 2/XL Module 54
//     Box 66 (AT5100-0100)/DRV Commutation angle/Commutation angle <-> Data Pointer/CommutationAngle
//     Box 66 (AT5100-0100)/DRV Controlword/Controlword <-> Data Pointer/Control
//     Box 66 (AT5100-0100)/DRV Statusword/Statusword <-> Data Pointer/Status
//     Box 66 (AT5100-0100)/DRV Target torque/Target torque <-> Data Pointer/Torque
//     Box 66 (AT5100-0100)/DRV Torque actual value/Torque actual value <-> Data Pointer/ActTorque
//     Box 66 (AT5100-0100)/XFB Inputs/Data <-> Data Pointer/HallSensorValues
//   (this object) <-> TcCOM Objects/XTS ProcessingUnit 1/XL Part 2/XL Module 55
//     Box 67 (AT5100-0100)/DRV Commutation angle/Commutation angle <-> Data Pointer/CommutationAngle
//     Box 67 (AT5100-0100)/DRV Controlword/Controlword <-> Data Pointer/Control
//     Box 67 (AT5100-0100)/DRV Statusword/Statusword <-> Data Pointer/Status
//     Box 67 (AT5100-0100)/DRV Target torque/Target torque <-> Data Pointer/Torque
//     Box 67 (AT5100-0100)/DRV Torque actual value/Torque actual value <-> Data Pointer/ActTorque
//     Box 67 (AT5100-0100)/XFB Inputs/Data <-> Data Pointer/HallSensorValues
//   (this object) <-> TcCOM Objects/XTS ProcessingUnit 1/XL Part 2/XL Module 56
//     Box 68 (AT5100-0100)/DRV Commutation angle/Commutation angle <-> Data Pointer/CommutationAngle
//     Box 68 (AT5100-0100)/DRV Controlword/Controlword <-> Data Pointer/Control
//     Box 68 (AT5100-0100)/DRV Statusword/Statusword <-> Data Pointer/Status
//     Box 68 (AT5100-0100)/DRV Target torque/Target torque <-> Data Pointer/Torque
//     Box 68 (AT5100-0100)/DRV Torque actual value/Torque actual value <-> Data Pointer/ActTorque
//     Box 68 (AT5100-0100)/XFB Inputs/Data <-> Data Pointer/HallSensorValues
//   (this object) <-> TcCOM Objects/XTS ProcessingUnit 1/XL Part 2/XL Module 57
//     Box 69 (AT5100-0100)/DRV Commutation angle/Commutation angle <-> Data Pointer/CommutationAngle
//     Box 69 (AT5100-0100)/DRV Controlword/Controlword <-> Data Pointer/Control
//     Box 69 (AT5100-0100)/DRV Statusword/Statusword <-> Data Pointer/Status
//     Box 69 (AT5100-0100)/DRV Target torque/Target torque <-> Data Pointer/Torque
//     Box 69 (AT5100-0100)/DRV Torque actual value/Torque actual value <-> Data Pointer/ActTorque
//     Box 69 (AT5100-0100)/XFB Inputs/Data <-> Data Pointer/HallSensorValues
//   (this object) <-> TcCOM Objects/XTS ProcessingUnit 1/Xl Part Start/XL Module 1
//     Box 74 (AT5100-0100)/DRV Commutation angle/Commutation angle <-> Data Pointer/CommutationAngle
//     Box 74 (AT5100-0100)/DRV Controlword/Controlword <-> Data Pointer/Control
//     Box 74 (AT5100-0100)/DRV Statusword/Statusword <-> Data Pointer/Status
//     Box 74 (AT5100-0100)/DRV Target torque/Target torque <-> Data Pointer/Torque
//     Box 74 (AT5100-0100)/DRV Torque actual value/Torque actual value <-> Data Pointer/ActTorque
//     Box 74 (AT5100-0100)/XFB Inputs/Data <-> Data Pointer/HallSensorValues
//   (this object) <-> TcCOM Objects/XTS ProcessingUnit 1/Xl Part Start/XL Module 2
//     Box 75 (AT5100-0100)/DRV Commutation angle/Commutation angle <-> Data Pointer/CommutationAngle
//     Box 75 (AT5100-0100)/DRV Controlword/Controlword <-> Data Pointer/Control
//     Box 75 (AT5100-0100)/DRV Statusword/Statusword <-> Data Pointer/Status
//     Box 75 (AT5100-0100)/DRV Target torque/Target torque <-> Data Pointer/Torque
//     Box 75 (AT5100-0100)/DRV Torque actual value/Torque actual value <-> Data Pointer/ActTorque
//     Box 75 (AT5100-0100)/XFB Inputs/Data <-> Data Pointer/HallSensorValues
//   (this object) <-> TcCOM Objects/XTS ProcessingUnit 1/Xl Part Start/XL Module 3
//     Box 76 (AT5100-0100)/DRV Commutation angle/Commutation angle <-> Data Pointer/CommutationAngle
//     Box 76 (AT5100-0100)/DRV Controlword/Controlword <-> Data Pointer/Control
//     Box 76 (AT5100-0100)/DRV Statusword/Statusword <-> Data Pointer/Status
//     Box 76 (AT5100-0100)/DRV Target torque/Target torque <-> Data Pointer/Torque
//     Box 76 (AT5100-0100)/DRV Torque actual value/Torque actual value <-> Data Pointer/ActTorque
//     Box 76 (AT5100-0100)/XFB Inputs/Data <-> Data Pointer/HallSensorValues
//   (this object) <-> TcCOM Objects/XTS ProcessingUnit 1/Xl Part Start/XL Module 46
//     Box 72 (AT5100-0100)/DRV Commutation angle/Commutation angle <-> Data Pointer/CommutationAngle
//     Box 72 (AT5100-0100)/DRV Controlword/Controlword <-> Data Pointer/Control
//     Box 72 (AT5100-0100)/DRV Statusword/Statusword <-> Data Pointer/Status
//     Box 72 (AT5100-0100)/DRV Target torque/Target torque <-> Data Pointer/Torque
//     Box 72 (AT5100-0100)/DRV Torque actual value/Torque actual value <-> Data Pointer/ActTorque
//     Box 72 (AT5100-0100)/XFB Inputs/Data <-> Data Pointer/HallSensorValues
//   (this object) <-> TcCOM Objects/XTS ProcessingUnit 1/Xl Part Start/XL Module 47
//     Box 73 (AT5100-0100)/DRV Commutation angle/Commutation angle <-> Data Pointer/CommutationAngle
//     Box 73 (AT5100-0100)/DRV Controlword/Controlword <-> Data Pointer/Control
//     Box 73 (AT5100-0100)/DRV Statusword/Statusword <-> Data Pointer/Status
//     Box 73 (AT5100-0100)/DRV Target torque/Target torque <-> Data Pointer/Torque
//     Box 73 (AT5100-0100)/DRV Torque actual value/Torque actual value <-> Data Pointer/ActTorque
//     Box 73 (AT5100-0100)/XFB Inputs/Data <-> Data Pointer/HallSensorValues
//   (this object) <-> MC Project IPC1/Groups/IPC 1 In Connection
//     Box 28 (Publisher)/MC Track - XL In Syst 1/Outputs/VarData <-> McToMc/ToNeighbourSystem
//     Box 29 (Subscriber)/MC Track - XL Out Syst 2/Inputs/VarData <-> McToMc/FromNeighbourSystem
//   (this object) <-> MC Project IPC1/Groups/IPC 1 Out Connection
//     Box 28 (Publisher)/MC Track - XL Out Syst 1/Outputs/VarData <-> McToMc/ToNeighbourSystem
//     Box 29 (Subscriber)/MC Track - XL In Syst 2/Inputs/VarData <-> McToMc/FromNeighbourSystem

// ---- DUTs/GVLs/GVL_IO.TcGVL

VAR_GLOBAL
	VoltageSet AT%Q*: REAL := 300;
	VoltageAct AT%I*: REAL;
	ControlDrive1121  AT%Q* : UINT;
	StatusDrive1121 AT%I* :UINT;
	ChargingResistor AT%Q* :BOOL;
	up , down : BOOL;
	start  : BOOL := TRUE;
	HwReset: BOOL;
	PowerSupplyReset AT%Q* : BOOL;
END_VAR

// ---- POUs/MAIN.TcPOU
PROGRAM MAIN
VAR
	nCase 					: INT;
	HwStart 		AT%I* 	: BOOL;
	HwStop  		AT%I* 	: BOOL;
	HwReset 		AT%I* 	: BOOL;
	xOn 			AT%Q* 	: BOOL;
	xRequestReset 	AT%Q* 	: BOOL;
	xError 			AT%Q* 	: BOOL;
		
	VoltageSP 			  	: LREAL := 300;
	rTrigSwitchon 		  	: R_trig;
	fTrigSwitchOff		  	: F_trig;
	Chargtimer 				: ton;
	
	SwitchOn				: BOOL;
	
	TcRestart :TC_Restart;
	Restart : BOOL;
	busy : BOOL;

END_VAR



IF GVL_Safety.HWStart OR hwstart THEN
	GVL_Safety.Run  := TRUE;
	GVL_Safety.Start := TRUE;
END_IF

IF  NOT GVL_Safety.HWStop THEN
	GVL_Safety.Run  := FALSE;
	GVL_Safety.Start := FALSE;
END_IF
		


IF gvl_safety.SaeftyOk THEN
	gvl_safety.HWSafetyOk := TRUE;
ELSE	
	gvl_safety.HWSafetyOk := FALSE;
END_IF

IF NOT gvl_safety.SafetyInRun THEN
	gvl_safety.HWerror := TRUE;
ELSE	
	gvl_safety.HWerror := FALSE;
END_IF

rTrigSwitchon(clk := HwStart );
fTrigSwitchOff(clk:= HwStop );


 Chargtimer(in := SwitchOn ,pt := T#1M, q=>GVL_IO.ChargingResistor);

IF rTrigSwitchon.Q THEN
	GVL_IO.VoltageSet := GVL_IO.VoltageAct;
	SwitchOn := TRUE;
ELSIF fTrigSwitchOff.Q THEN
	SwitchOn := FALSE;
	GVL_IO.VoltageSet :=   0;
END_IF



IF (VoltageSP-2) > GVL_IO.VoltageAct AND  GVL_IO.Voltageset <VoltageSP AND SwitchOn THEN
	GVL_IO.VoltageSet := GVL_IO.VoltageSet +0.1;
END_IF



IF GVL_IO.hwReset OR HwReset THEN
	GVL_IO.ControlDrive1121 := 16#FF;
	GVL_Safety.Reset := TRUE;
	GVL_IO.PowerSupplyReset := TRUE;
ELSE 	
	GVL_IO.ControlDrive1121 := 16#0;
	GVL_Safety.Reset := FALSE;
	GVL_IO.PowerSupplyReset := FALSE;
END_IF


TcRestart(
	NETID:= , 
	RESTART:=Restart , 
	TMOUT:= , 
	BUSY=> , 
	ERR=> , 
	ERRID=> );

END_PROGRAM
